fbVoter1Button(stColor := fbVoter1.fbStatusColor, nActiveTab := eActiveTab, sActiveName := sActiveName);
fbVoter2Button(stColor := fbVoter2.fbStatusColor, nActiveTab := eActiveTab, sActiveName := sActiveName);
fbVoter3Button(stColor := fbVoter3.fbStatusColor, nActiveTab := eActiveTab, sActiveName := sActiveName);
fbVoter4Button(stColor := fbVoter4.fbStatusColor, nActiveTab := eActiveTab, sActiveName := sActiveName);
fbVoter5Button(stColor := fbVoter5.fbStatusColor, nActiveTab := eActiveTab, sActiveName := sActiveName);
fbVoter6Button(stColor := fbVoter6.fbStatusColor, nActiveTab := eActiveTab, sActiveName := sActiveName);
fbVoter7Button(stColor := fbVoter7.fbStatusColor, nActiveTab := eActiveTab, sActiveName := sActiveName);
fbVoter8Button(stColor := fbVoter8.fbStatusColor, nActiveTab := eActiveTab, sActiveName := sActiveName);
fbVoter9Button(stColor := fbVoter9.fbStatusColor, nActiveTab := eActiveTab, sActiveName := sActiveName);
fbVoter10Button(stColor := fbVoter10.fbStatusColor, nActiveTab := eActiveTab, sActiveName := sActiveName);
    
M_UpdateStatusColor();

END_FUNCTION_BLOCK

// HMI/POUs/Subsystems/IMG/FB_HMI_IMG
FUNCTION_BLOCK FB_HMI_IMG EXTENDS FB_HMI_COMPONENT
VAR_INPUT
    bConnected : BOOL;
END_VAR
VAR_OUTPUT
END_VAR
VAR_IN_OUT
    temperatures    : FB_METIS_TEMPERATURES;
    heaters         : FB_METIS_HEATERS;
    voters          : FB_METIS_VOTERS;
    tctrl           : FB_METIS_TCTRL;
    lakeshores      : FB_METIS_LAKESHORES;
END_VAR
VAR
    // active tab of the main frame
    eActiveTab : E_HMI_IMG_TABS := E_HMI_IMG_TABS.TEMPERATURES;
    sActiveName : STRING;
    
    // components
    fbTemperatures : FB_HMI_IMG_TEMPERATURES;
    fbVoters       : FB_HMI_IMG_VOTERS;
    fbTControl     : FB_HMI_IMG_TCTRL;
    fbHeaters      : FB_HMI_IMG_HEATERS;
    fbLakeshoreLm  : FB_HMI_LAKESHORE;
    fbLakeshoreN   : FB_HMI_LAKESHORE;
    
    // buttons
    fbTemperaturesButton : FB_HMI_BUTTON(sName := 'Temperatures'         , sIconName := '', nThisTab := E_HMI_IMG_TABS.TEMPERATURES);
    fbVotersButton       : FB_HMI_BUTTON(sName := 'Voters'               , sIconName := '', nThisTab := E_HMI_IMG_TABS.VOTERS);
    fbHeatersButton      : FB_HMI_BUTTON(sName := 'Heaters'              , sIconName := '', nThisTab := E_HMI_IMG_TABS.HEATERS);
    fbLakeshoreLmButton  : FB_HMI_BUTTON(sName := 'Lakeshore LM'         , sIconName := '', nThisTab := E_HMI_IMG_TABS.LAKESHORE_LM_DET);
    fbLakeshoreNButton   : FB_HMI_BUTTON(sName := 'Lakeshore N'          , sIconName := '', nThisTab := E_HMI_IMG_TABS.LAKESHORE_N_DET);
    fbTControlButton     : FB_HMI_BUTTON(sName := 'Control loops'        , sIconName := '', nThisTab := E_HMI_IMG_TABS.TCONTROL);
    
    // connection status
    sConnected           : STRING;
    eConnectedColor      : E_HMI_COLORS;
END_VAR

// update the connection status
sConnected      := F_GetConnectionString(bConnected);
eConnectedColor := F_GetConnectionColor(bConnected); 

// update the components
fbTemperatures(fbInstance := temperatures, bConnected := bConnected);
fbVoters(fbInstance := voters, bConnected := bConnected);
fbTControl(fbInstance := tctrl, bConnected := bConnected);
fbHeaters(fbInstance := heaters, bConnected := bConnected);
fbLakeshoreLm(fbInstance := lakeshores.ls_img_lm, bConnected := bConnected);
fbLakeshoreN(fbInstance := lakeshores.ls_img_n, bConnected := bConnected);


// update the buttons
// sca
fbTemperaturesButton(
    stColor     := fbTemperatures.fbStatusColor,
    nActiveTab  := eActiveTab,
    sActiveName := sActiveName);
fbVotersButton(
    stColor     := fbVoters.fbStatusColor,
    nActiveTab  := eActiveTab,
    sActiveName := sActiveName);
fbHeatersButton(
    stColor     := fbHeaters.fbStatusColor,
    nActiveTab  := eActiveTab,
    sActiveName := sActiveName);
fbLakeshoreLmButton(
    stColor     := fbLakeshoreLm.fbStatusColor,
    nActiveTab  := eActiveTab,
    sActiveName := sActiveName);
fbLakeshoreNButton(
    stColor     := fbLakeshoreN.fbStatusColor,
    nActiveTab  := eActiveTab,
    sActiveName := sActiveName);
fbTControlButton(
    stColor     := fbTControl.fbStatusColor,
    nActiveTab  := eActiveTab,
    sActiveName := sActiveName);

// update the summary health/busy status
fbHealthStatus(
    bIsEnabled  := bConnected,
    bIsGood     :=     fbTemperatures.fbHealthStatus.bGood
                   AND fbVoters.fbHealthStatus.bGood
                   AND fbTControl.fbHealthStatus.bGood
                   AND fbHeaters.fbHealthStatus.bGood
                   AND fbLakeshoreLm.fbHealthStatus.bGood
                   AND fbLakeshoreN.fbHealthStatus.bGood,
    bHasWarning :=     fbTemperatures.fbHealthStatus.bWarning
                    OR fbVoters.fbHealthStatus.bWarning
                    OR fbTControl.fbHealthStatus.bWarning
                    OR fbHeaters.fbHealthStatus.bWarning
                    OR fbLakeshoreLm.fbHealthStatus.bWarning
                    OR fbLakeshoreN.fbHealthStatus.bWarning);

fbBusyStatus(
    bIsEnabled   := bConnected,
    bIsBusy      :=    fbTemperatures.fbBusyStatus.bBusy
                    OR fbVoters.fbBusyStatus.bBusy
                    OR fbTControl.fbBusyStatus.bBusy
                    OR fbHeaters.fbBusyStatus.bBusy
                    OR fbLakeshoreLm.fbBusyStatus.bBusy
                    OR fbLakeshoreN.fbBusyStatus.bBusy);

M_UpdateStatusColor();

END_FUNCTION_BLOCK

// HMI/POUs/Util/Functions/F_GetConnectionString
FUNCTION F_GetConnectionString : STRING
VAR_INPUT
    bConnected : BOOL;
END_VAR
VAR
END_VAR

IF bConnected THEN
    F_GetConnectionString := 'Connected';
ELSE
    F_GetConnectionString := 'Disconnected';
END_IF

END_FUNCTION

// HMI/POUs/Util/Functions/F_GetConnectionColor
FUNCTION F_GetConnectionColor : E_HMI_COLORS
VAR_INPUT
    bConnected : BOOL;
END_VAR
VAR
END_VAR

IF bConnected THEN
    F_GetConnectionColor := E_HMI_COLORS.GREEN;
ELSE
    F_GetConnectionColor := E_HMI_COLORS.RED;
END_IF

END_FUNCTION

// HMI/POUs/Subsystems/LMS/Components/FB_HMI_LMS_HEATERS
FUNCTION_BLOCK FB_HMI_LMS_HEATERS EXTENDS FB_HMI_COMPONENT
VAR_INPUT
END_VAR
VAR_OUTPUT
END_VAR
VAR_IN_OUT
    fbInstance : FB_METIS_HEATERS;
END_VAR
VAR
//    eActiveTab : E_HMI_CRY_HEATER_TABS;
//    sActiveName : STRING;
    
//    h_img_wuh_1_button  : FB_HMI_BUTTON(sName := 'H_IMG_WUH_1' , sIconName := '', nThisTab := E_HMI_IMG_HEATER_TABS.H_IMG_WUH_1);
//    h_img_wuh_2_button  : FB_HMI_BUTTON(sName := 'H_IMG_WUH_2' , sIconName := '', nThisTab := E_HMI_IMG_HEATER_TABS.H_IMG_WUH_2);
//    h_img_lmd_2_button  : FB_HMI_BUTTON(sName := 'H_IMG_LMD_2' , sIconName := '', nThisTab := E_HMI_IMG_HEATER_TABS.H_IMG_LMD_2);
//    h_img_lmp_2_button  : FB_HMI_BUTTON(sName := 'H_IMG_LMP_2' , sIconName := '', nThisTab := E_HMI_IMG_HEATER_TABS.H_IMG_LMP_2);
//    h_img_nd_2_button   : FB_HMI_BUTTON(sName := 'H_IMG_ND_2'  , sIconName := '', nThisTab := E_HMI_IMG_HEATER_TABS.H_IMG_ND_2);
    
//    h_img_wuh_1 : FB_HMI_METIS_HEATER;
//    h_img_wuh_2 : FB_HMI_METIS_HEATER;
//    h_img_lmd_2 : FB_HMI_METIS_HEATER;
//    h_img_lmp_2 : FB_HMI_METIS_HEATER;
//    h_img_nd_2  : FB_HMI_METIS_HEATER;
END_VAR

fbHealthStatus(bIsEnabled := FALSE);
fbBusyStatus(bIsEnabled := FALSE);

//fbHealthStatus(
//    bIsEnabled := TRUE,
//    bIsGood := NOT(    fbInstance.h_img_wuh_1.stat.bError
//                    OR fbInstance.h_img_wuh_2.stat.bError
//                    OR fbInstance.h_img_lmd_2.stat.bError
//                    OR fbInstance.h_img_lmp_2.stat.bError
//                    OR fbInstance.h_img_nd_2.stat.bError ),
//    bHasWarning := (    fbInstance.h_img_wuh_1.stat.bWarning
//                     OR fbInstance.h_img_wuh_2.stat.bWarning
//                     OR fbInstance.h_img_lmd_2.stat.bWarning
//                     OR fbInstance.h_img_lmp_2.stat.bWarning
//                     OR fbInstance.h_img_nd_2.stat.bWarning));

//fbBusyStatus(
//    bIsEnabled := TRUE,
//    bIsBusy := FALSE);

//h_img_wuh_1(fbInstance := fbInstance.h_img_wuh_1);
//h_img_wuh_2(fbInstance := fbInstance.h_img_wuh_2);
//h_img_lmd_2(fbInstance := fbInstance.h_img_lmd_2);
//h_img_lmp_2(fbInstance := fbInstance.h_img_lmp_2);
//h_img_nd_2(fbInstance := fbInstance.h_img_nd_2);

//h_img_wuh_1_button(stColor := h_img_wuh_1.fbStatusColor, nActiveTab := eActiveTab, sActiveName := sActiveName);
//h_img_wuh_2_button(stColor := h_img_wuh_2.fbStatusColor, nActiveTab := eActiveTab, sActiveName := sActiveName);
//h_img_lmd_2_button(stColor := h_img_lmd_2.fbStatusColor, nActiveTab := eActiveTab, sActiveName := sActiveName);
//h_img_lmp_2_button(stColor := h_img_lmp_2.fbStatusColor, nActiveTab := eActiveTab, sActiveName := sActiveName);
//h_img_nd_2_button(stColor := h_img_nd_2.fbStatusColor, nActiveTab := eActiveTab, sActiveName := sActiveName);

M_UpdateStatusColor();

END_FUNCTION_BLOCK

// HMI/POUs/Subsystems/LMS/Components/FB_HMI_LMS_TCTRL
FUNCTION_BLOCK FB_HMI_LMS_TCTRL EXTENDS FB_HMI_COMPONENT
VAR_INPUT
END_VAR
VAR_OUTPUT
END_VAR
VAR_IN_OUT
    fbInstance : FB_METIS_TCTRL;
END_VAR
VAR
//    eActiveTab : E_HMI_IMG_TC_TABS;
//    sActiveName : STRING;
    
//    tc_img_wuh_1_button  : FB_HMI_BUTTON(sName := 'TC_IMG_WUH_1' , sIconName := '', nThisTab := E_HMI_IMG_TC_TABS.TC_IMG_WUH_1);
//    tc_img_wuh_2_button  : FB_HMI_BUTTON(sName := 'TC_IMG_WUH_2' , sIconName := '', nThisTab := E_HMI_IMG_TC_TABS.TC_IMG_WUH_2);
//    tc_img_lmd_2_button  : FB_HMI_BUTTON(sName := 'TC_IMG_LMD_2' , sIconName := '', nThisTab := E_HMI_IMG_TC_TABS.TC_IMG_LMD_2);
//    tc_img_lmp_2_button  : FB_HMI_BUTTON(sName := 'TC_IMG_LMP_2' , sIconName := '', nThisTab := E_HMI_IMG_TC_TABS.TC_IMG_LMP_2);
//    tc_img_nd_2_button   : FB_HMI_BUTTON(sName := 'TC_IMG_ND_2'  , sIconName := '', nThisTab := E_HMI_IMG_TC_TABS.TC_IMG_ND_2);
    
//    tc_img_wuh_1 : FB_HMI_METIS_CTRL_DT670;
//    tc_img_wuh_2 : FB_HMI_METIS_CTRL_DT670;
//    tc_img_lmd_2 : FB_HMI_METIS_CTRL_DT670;
//    tc_img_lmp_2 : FB_HMI_METIS_CTRL_DT670;
//    tc_img_nd_2  : FB_HMI_METIS_CTRL_DT670;
END_VAR

fbHealthStatus(bIsEnabled := FALSE);
fbBusyStatus(bIsEnabled := FALSE);

//fbHealthStatus(
//    bIsEnabled := TRUE,
//    bIsGood := NOT(    fbInstance.tc_img_wuh_1.stat.bError
//                    OR fbInstance.tc_img_wuh_2.stat.bError
//                    OR fbInstance.tc_img_lmd_2.stat.bError
//                    OR fbInstance.tc_img_lmp_2.stat.bError
//                    OR fbInstance.tc_img_nd_2.stat.bError ),
//    bHasWarning := (    fbInstance.tc_img_wuh_1.stat.bWarning
//                     OR fbInstance.tc_img_wuh_2.stat.bWarning
//                     OR fbInstance.tc_img_lmd_2.stat.bWarning
//                     OR fbInstance.tc_img_lmp_2.stat.bWarning
//                     OR fbInstance.tc_img_nd_2.stat.bWarning));

//tc_img_wuh_1(fbInstance := fbInstance.tc_img_wuh_1);
//tc_img_wuh_2(fbInstance := fbInstance.tc_img_wuh_2);
//tc_img_lmd_2(fbInstance := fbInstance.tc_img_lmd_2);
//tc_img_lmp_2(fbInstance := fbInstance.tc_img_lmp_2);
//tc_img_nd_2(fbInstance := fbInstance.tc_img_nd_2);

//tc_img_wuh_1_button(stColor := tc_img_wuh_1.fbStatusColor, nActiveTab := eActiveTab, sActiveName := sActiveName);
//tc_img_wuh_2_button(stColor := tc_img_wuh_2.fbStatusColor, nActiveTab := eActiveTab, sActiveName := sActiveName);
//tc_img_lmd_2_button(stColor := tc_img_lmd_2.fbStatusColor, nActiveTab := eActiveTab, sActiveName := sActiveName);
//tc_img_lmp_2_button(stColor := tc_img_lmp_2.fbStatusColor, nActiveTab := eActiveTab, sActiveName := sActiveName);
//tc_img_nd_2_button(stColor := tc_img_nd_2.fbStatusColor, nActiveTab := eActiveTab, sActiveName := sActiveName);

//fbBusyStatus(
//    bIsEnabled := TRUE,
//    bIsBusy := FALSE);

M_UpdateStatusColor();

END_FUNCTION_BLOCK

// HMI/POUs/Subsystems/LMS/Components/FB_HMI_LMS_TEMPERATURES
FUNCTION_BLOCK FB_HMI_LMS_TEMPERATURES EXTENDS FB_HMI_COMPONENT
VAR_INPUT
END_VAR
VAR_OUTPUT
END_VAR
VAR_IN_OUT
    fbInstance : FB_METIS_TEMPERATURES;
END_VAR
VAR
END_VAR

fbHealthStatus(bIsEnabled := FALSE);
fbBusyStatus(bIsEnabled := FALSE);

//fbHealthStatus(
//    bIsEnabled := TRUE,
//    bIsGood :=     fbInstance.t_img_lpw_1.stat.bValid
//               AND fbInstance.t_img_lpw_2.stat.bValid
//               AND fbInstance.t_img_lfw_1.stat.bValid
//               AND fbInstance.t_img_lfw_2.stat.bValid
//               AND fbInstance.t_img_lpr_1.stat.bValid
//               AND fbInstance.t_img_bwu_3.stat.bValid
//               AND fbInstance.t_img_lnd_1.stat.bValid
//               AND fbInstance.t_img_lnd_2.stat.bValid
//               AND fbInstance.t_img_npw_1.stat.bValid
//               AND fbInstance.t_img_npw_2.stat.bValid
//               AND fbInstance.t_img_nfw_1.stat.bValid
//               AND fbInstance.t_img_nfw_2.stat.bValid
//               AND fbInstance.t_img_npr_1.stat.bValid
//               AND fbInstance.t_img_bwu_2.stat.bValid
//               AND fbInstance.t_img_nnd_1.stat.bValid
//               AND fbInstance.t_img_nnd_2.stat.bValid
//               AND fbInstance.t_img_opt_1.stat.bValid
//               AND fbInstance.t_img_bwu_1.stat.bValid
//               AND fbInstance.t_img_ctr_1.stat.bValid
//               AND fbInstance.t_img_ctr_2.stat.bValid
//               AND fbInstance.t_img_70k_1.stat.bValid
//               AND fbInstance.t_img_ln2_1.stat.bValid
//               AND fbInstance.t_img_ln2_2.stat.bValid
//               AND fbInstance.t_img_hex_1.stat.bValid
//               AND fbInstance.t_img_lmd_1.stat.bValid
//               AND fbInstance.t_img_lmd_2.stat.bValid
//               AND fbInstance.t_img_lmp_1.stat.bValid
//               AND fbInstance.t_img_lmp_2.stat.bValid
//               AND fbInstance.t_img_nd_1.stat.bValid
//               AND fbInstance.t_img_nd_2.stat.bValid,
//    bHasWarning := (    fbInstance.t_img_lpw_1.stat.bWarning
//                     OR fbInstance.t_img_lpw_2.stat.bWarning
//                     OR fbInstance.t_img_lfw_1.stat.bWarning
//                     OR fbInstance.t_img_lfw_2.stat.bWarning
//                     OR fbInstance.t_img_lpr_1.stat.bWarning
//                     OR fbInstance.t_img_bwu_3.stat.bWarning
//                     OR fbInstance.t_img_lnd_1.stat.bWarning
//                     OR fbInstance.t_img_lnd_2.stat.bWarning
//                     OR fbInstance.t_img_npw_1.stat.bWarning
//                     OR fbInstance.t_img_npw_2.stat.bWarning
//                     OR fbInstance.t_img_nfw_1.stat.bWarning
//                     OR fbInstance.t_img_nfw_2.stat.bWarning
//                     OR fbInstance.t_img_npr_1.stat.bWarning
//                     OR fbInstance.t_img_bwu_2.stat.bWarning
//                     OR fbInstance.t_img_nnd_1.stat.bWarning
//                     OR fbInstance.t_img_nnd_2.stat.bWarning
//                     OR fbInstance.t_img_opt_1.stat.bWarning
//                     OR fbInstance.t_img_bwu_1.stat.bWarning
//                     OR fbInstance.t_img_ctr_1.stat.bWarning
//                     OR fbInstance.t_img_ctr_2.stat.bWarning
//                     OR fbInstance.t_img_ln2_1.stat.bWarning
//                     OR fbInstance.t_img_ln2_1.stat.bWarning
//                     OR fbInstance.t_img_ln2_2.stat.bWarning
//                     OR fbInstance.t_img_hex_1.stat.bWarning
//                     OR fbInstance.t_img_lmd_1.stat.bWarning
//                     OR fbInstance.t_img_lmd_2.stat.bWarning
//                     OR fbInstance.t_img_lmp_1.stat.bWarning
//                     OR fbInstance.t_img_lmp_2.stat.bWarning
//                     OR fbInstance.t_img_nd_1.stat.bWarning
//                     OR fbInstance.t_img_nd_2.stat.bWarning));
                     
//fbBusyStatus(
//    bIsEnabled := TRUE,
//    bIsBusy := FALSE);

M_UpdateStatusColor();

END_FUNCTION_BLOCK

// HMI/POUs/Subsystems/LMS/Components/FB_HMI_LMS_VOTERS
FUNCTION_BLOCK FB_HMI_LMS_VOTERS EXTENDS FB_HMI_COMPONENT
VAR_INPUT
END_VAR
VAR_OUTPUT
END_VAR
VAR_IN_OUT
    fbInstance : FB_METIS_VOTERS;
END_VAR
VAR
    eActiveTab : E_HMI_VOTER_TABS;
    sActiveName : STRING;
    
    fbVoter1Button  : FB_HMI_BUTTON(sName := 'Voter 1' , sIconName := '', nThisTab := E_HMI_VOTER_TABS.VOTER_1);
    fbVoter2Button  : FB_HMI_BUTTON(sName := 'Voter 2' , sIconName := '', nThisTab := E_HMI_VOTER_TABS.VOTER_2);
    fbVoter3Button  : FB_HMI_BUTTON(sName := 'Voter 3' , sIconName := '', nThisTab := E_HMI_VOTER_TABS.VOTER_3);
    fbVoter4Button  : FB_HMI_BUTTON(sName := 'Voter 4' , sIconName := '', nThisTab := E_HMI_VOTER_TABS.VOTER_4);
    fbVoter5Button  : FB_HMI_BUTTON(sName := 'Voter 5' , sIconName := '', nThisTab := E_HMI_VOTER_TABS.VOTER_5);
    fbVoter6Button  : FB_HMI_BUTTON(sName := 'Voter 6' , sIconName := '', nThisTab := E_HMI_VOTER_TABS.VOTER_6);
    fbVoter7Button  : FB_HMI_BUTTON(sName := 'Voter 7' , sIconName := '', nThisTab := E_HMI_VOTER_TABS.VOTER_7);
    fbVoter8Button  : FB_HMI_BUTTON(sName := 'Voter 8' , sIconName := '', nThisTab := E_HMI_VOTER_TABS.VOTER_8);
    fbVoter9Button  : FB_HMI_BUTTON(sName := 'Voter 9' , sIconName := '', nThisTab := E_HMI_VOTER_TABS.VOTER_9);
    fbVoter10Button : FB_HMI_BUTTON(sName := 'Voter 10', sIconName := '', nThisTab := E_HMI_VOTER_TABS.VOTER_10);
    
    fbVoter1 : FB_HMI_VOTER;
    fbVoter2 : FB_HMI_VOTER;
    fbVoter3 : FB_HMI_VOTER;
    fbVoter4 : FB_HMI_VOTER;
    fbVoter5 : FB_HMI_VOTER;
    fbVoter6 : FB_HMI_VOTER;
    fbVoter7 : FB_HMI_VOTER;
    fbVoter8 : FB_HMI_VOTER;
    fbVoter9 : FB_HMI_VOTER;
    fbVoter10 : FB_HMI_VOTER;
END_VAR

fbHealthStatus(bIsEnabled := FALSE);
fbBusyStatus(bIsEnabled := FALSE);

//fbHealthStatus(
//    bIsEnabled :=  fbVoter1.fbHealthStatus.bEnabled
//                OR fbVoter2.fbHealthStatus.bEnabled
//                OR fbVoter3.fbHealthStatus.bEnabled
//                OR fbVoter4.fbHealthStatus.bEnabled
//                OR fbVoter5.fbHealthStatus.bEnabled
//                OR fbVoter6.fbHealthStatus.bEnabled
//                OR fbVoter7.fbHealthStatus.bEnabled
//                OR fbVoter8.fbHealthStatus.bEnabled
//                OR fbVoter9.fbHealthStatus.bEnabled
//                OR fbVoter10.fbHealthStatus.bEnabled,
//    bIsGood :=  (fbVoter1.fbHealthStatus.bGood OR NOT fbVoter1.fbHealthStatus.bEnabled)
//            AND (fbVoter2.fbHealthStatus.bGood OR NOT fbVoter2.fbHealthStatus.bEnabled)
//            AND (fbVoter3.fbHealthStatus.bGood OR NOT fbVoter3.fbHealthStatus.bEnabled)
//            AND (fbVoter4.fbHealthStatus.bGood OR NOT fbVoter4.fbHealthStatus.bEnabled)
//            AND (fbVoter5.fbHealthStatus.bGood OR NOT fbVoter5.fbHealthStatus.bEnabled)
//            AND (fbVoter6.fbHealthStatus.bGood OR NOT fbVoter6.fbHealthStatus.bEnabled)
//            AND (fbVoter7.fbHealthStatus.bGood OR NOT fbVoter7.fbHealthStatus.bEnabled)
//            AND (fbVoter8.fbHealthStatus.bGood OR NOT fbVoter8.fbHealthStatus.bEnabled)
//            AND (fbVoter9.fbHealthStatus.bGood OR NOT fbVoter9.fbHealthStatus.bEnabled)
//            AND (fbVoter10.fbHealthStatus.bGood OR NOT fbVoter10.fbHealthStatus.bEnabled));

//fbBusyStatus(
//    bIsEnabled := TRUE,
//    bIsBusy := FALSE);

//fbVoter1(fbInstance := fbInstance.vote_img_1);
//fbVoter2(fbInstance := fbInstance.vote_img_2);
//fbVoter3(fbInstance := fbInstance.vote_img_3);
//fbVoter4(fbInstance := fbInstance.vote_img_4);
//fbVoter5(fbInstance := fbInstance.vote_img_5);
//fbVoter6(fbInstance := fbInstance.vote_img_6);
//fbVoter7(fbInstance := fbInstance.vote_img_7);
//fbVoter8(fbInstance := fbInstance.vote_img_8);
//fbVoter9(fbInstance := fbInstance.vote_img_9);
//fbVoter10(fbInstance := fbInstance.vote_img_10);

//fbVoter1Button(stColor := fbVoter1.fbStatusColor, nActiveTab := eActiveTab, sActiveName := sActiveName);
//fbVoter2Button(stColor := fbVoter2.fbStatusColor, nActiveTab := eActiveTab, sActiveName := sActiveName);
//fbVoter3Button(stColor := fbVoter3.fbStatusColor, nActiveTab := eActiveTab, sActiveName := sActiveName);
//fbVoter4Button(stColor := fbVoter4.fbStatusColor, nActiveTab := eActiveTab, sActiveName := sActiveName);
//fbVoter5Button(stColor := fbVoter5.fbStatusColor, nActiveTab := eActiveTab, sActiveName := sActiveName);
//fbVoter6Button(stColor := fbVoter6.fbStatusColor, nActiveTab := eActiveTab, sActiveName := sActiveName);
//fbVoter7Button(stColor := fbVoter7.fbStatusColor, nActiveTab := eActiveTab, sActiveName := sActiveName);
//fbVoter8Button(stColor := fbVoter8.fbStatusColor, nActiveTab := eActiveTab, sActiveName := sActiveName);
//fbVoter9Button(stColor := fbVoter9.fbStatusColor, nActiveTab := eActiveTab, sActiveName := sActiveName);
//fbVoter10Button(stColor := fbVoter10.fbStatusColor, nActiveTab := eActiveTab, sActiveName := sActiveName);
    
M_UpdateStatusColor();

END_FUNCTION_BLOCK

// HMI/POUs/Subsystems/LMS/FB_HMI_LMS
FUNCTION_BLOCK FB_HMI_LMS EXTENDS FB_HMI_COMPONENT
VAR_INPUT
END_VAR
VAR_OUTPUT
END_VAR
VAR_IN_OUT
    temperatures    : FB_METIS_TEMPERATURES;
    heaters         : FB_METIS_HEATERS;
    voters          : FB_METIS_VOTERS;
    tctrl           : FB_METIS_TCTRL;
END_VAR
VAR
    // active tab of the main frame
    eActiveTab : E_HMI_LMS_TABS := E_HMI_LMS_TABS.TEMPERATURES;
    sActiveName : STRING;
    
    // components
    fbTemperatures : FB_HMI_LMS_TEMPERATURES;
    fbVoters       : FB_HMI_LMS_VOTERS;
    fbTControl     : FB_HMI_LMS_TCTRL;
    fbHeaters      : FB_HMI_LMS_HEATERS;
    
    // buttons
    fbTemperaturesButton : FB_HMI_BUTTON(sName := 'Temperatures'         , sIconName := '', nThisTab := E_HMI_LMS_TABS.TEMPERATURES);
    fbVotersButton       : FB_HMI_BUTTON(sName := 'Voters'               , sIconName := '', nThisTab := E_HMI_LMS_TABS.VOTERS);
    fbHeatersButton      : FB_HMI_BUTTON(sName := 'Heaters'              , sIconName := '', nThisTab := E_HMI_LMS_TABS.HEATERS);
    fbTControlButton     : FB_HMI_BUTTON(sName := 'Control loops'        , sIconName := '', nThisTab := E_HMI_LMS_TABS.TCONTROL);
END_VAR

// update the components
fbTemperatures(fbInstance := temperatures);
fbVoters(fbInstance := voters);
fbTControl(fbInstance := tctrl);
fbHeaters(fbInstance := heaters);

// update the buttons
fbTemperaturesButton(
    stColor     := fbTemperatures.fbStatusColor,
    nActiveTab  := eActiveTab,
    sActiveName := sActiveName);
fbVotersButton(
    stColor     := fbVoters.fbStatusColor,
    nActiveTab  := eActiveTab,
    sActiveName := sActiveName);
fbHeatersButton(
    stColor     := fbHeaters.fbStatusColor,
    nActiveTab  := eActiveTab,
    sActiveName := sActiveName);
fbTControlButton(
    stColor     := fbTControl.fbStatusColor,
    nActiveTab  := eActiveTab,
    sActiveName := sActiveName);


// update the summary health/busy status
fbHealthStatus(
    bIsEnabled  := TRUE,
    bIsGood     :=     fbTemperatures.fbHealthStatus.bGood
                   AND fbVoters.fbHealthStatus.bGood
                   AND fbTControl.fbHealthStatus.bGood
                   AND fbHeaters.fbHealthStatus.bGood,
    bHasWarning :=     fbTemperatures.fbHealthStatus.bWarning
                    OR fbVoters.fbHealthStatus.bWarning
                    OR fbTControl.fbHealthStatus.bWarning
                    OR fbHeaters.fbHealthStatus.bWarning);

fbBusyStatus(
    bIsEnabled   := TRUE,
    bIsBusy      :=    fbTemperatures.fbBusyStatus.bBusy
                    OR fbVoters.fbBusyStatus.bBusy
                    OR fbTControl.fbBusyStatus.bBusy
                    OR fbHeaters.fbBusyStatus.bBusy);

M_UpdateStatusColor();

END_FUNCTION_BLOCK

// HMI/POUs/Subsystems/SCA/Components/FB_HMI_SCA_HEATERS
FUNCTION_BLOCK FB_HMI_SCA_HEATERS EXTENDS FB_HMI_COMPONENT
VAR_INPUT
    bConnected : BOOL;
END_VAR
VAR_OUTPUT
END_VAR
VAR_IN_OUT
    fbInstance : FB_METIS_HEATERS;
END_VAR
VAR
    eActiveTab : E_HMI_SCA_HEATER_TABS;
    sActiveName : STRING;
    
    h_sca_wuh_1_button  : FB_HMI_BUTTON(sName := 'H_SCA_WUH_1' , sIconName := '', nThisTab := E_HMI_SCA_HEATER_TABS.H_SCA_WUH_1);
    h_sca_wuh_2_button  : FB_HMI_BUTTON(sName := 'H_SCA_WUH_2' , sIconName := '', nThisTab := E_HMI_SCA_HEATER_TABS.H_SCA_WUH_2);
    h_sca_det_2_button  : FB_HMI_BUTTON(sName := 'H_SCA_DET_2' , sIconName := '', nThisTab := E_HMI_SCA_HEATER_TABS.H_SCA_DET_2);
    h_sca_dhs_2_button  : FB_HMI_BUTTON(sName := 'H_SCA_DHS_2' , sIconName := '', nThisTab := E_HMI_SCA_HEATER_TABS.H_SCA_DHS_2);
    
    h_sca_wuh_1 : FB_HMI_METIS_HEATER;
    h_sca_wuh_2 : FB_HMI_METIS_HEATER;
    h_sca_det_2 : FB_HMI_METIS_HEATER;
    h_sca_dhs_2 : FB_HMI_METIS_HEATER;
END_VAR

fbHealthStatus(
    bIsEnabled := bConnected,
    bIsGood := NOT(    fbInstance.h_sca_wuh_1.stat.bError
                    OR fbInstance.h_sca_wuh_2.stat.bError
                    OR fbInstance.h_sca_det_2.stat.bError
                    OR fbInstance.h_sca_dhs_2.stat.bError ),
    bHasWarning := (    fbInstance.h_sca_wuh_1.stat.bWarning
                     OR fbInstance.h_sca_wuh_2.stat.bWarning
                     OR fbInstance.h_sca_det_2.stat.bWarning
                     OR fbInstance.h_sca_dhs_2.stat.bWarning));
                     
fbBusyStatus(
    bIsEnabled := bConnected,
    bIsBusy := FALSE);

h_sca_wuh_1(fbInstance := fbInstance.h_sca_wuh_1);
h_sca_wuh_2(fbInstance := fbInstance.h_sca_wuh_2);
h_sca_det_2(fbInstance := fbInstance.h_sca_det_2);
h_sca_dhs_2(fbInstance := fbInstance.h_sca_dhs_2);

h_sca_wuh_1_button(stColor := h_sca_wuh_1.fbStatusColor, nActiveTab := eActiveTab, sActiveName := sActiveName);
h_sca_wuh_2_button(stColor := h_sca_wuh_2.fbStatusColor, nActiveTab := eActiveTab, sActiveName := sActiveName);
h_sca_det_2_button(stColor := h_sca_det_2.fbStatusColor, nActiveTab := eActiveTab, sActiveName := sActiveName);
h_sca_dhs_2_button(stColor := h_sca_dhs_2.fbStatusColor, nActiveTab := eActiveTab, sActiveName := sActiveName);

M_UpdateStatusColor();

END_FUNCTION_BLOCK

// HMI/POUs/Subsystems/SCA/Components/FB_HMI_SCA_TCTRL
FUNCTION_BLOCK FB_HMI_SCA_TCTRL EXTENDS FB_HMI_COMPONENT
VAR_INPUT
    bConnected : BOOL;
END_VAR
VAR_OUTPUT
END_VAR
VAR_IN_OUT
    fbInstance : FB_METIS_TCTRL;
END_VAR
VAR
    eActiveTab : E_HMI_SCA_TC_TABS;
    sActiveName : STRING;
    
    tc_sca_wuh_button    : FB_HMI_BUTTON(sName := 'TC_SCA_WUH'   , sIconName := '', nThisTab := E_HMI_SCA_TC_TABS.TC_SCA_WUH);
    tc_sca_det_2_button  : FB_HMI_BUTTON(sName := 'TC_SCA_DET_2' , sIconName := '', nThisTab := E_HMI_SCA_TC_TABS.TC_SCA_DET_2);
    tc_sca_dhs_2_button  : FB_HMI_BUTTON(sName := 'TC_SCA_DHS_2' , sIconName := '', nThisTab := E_HMI_SCA_TC_TABS.TC_SCA_DHS_2);
    
    tc_sca_wuh   : FB_HMI_METIS_CTRL_TEMPERATURE;
    tc_sca_det_2 : FB_HMI_METIS_CTRL_TEMPERATURE;
    tc_sca_dhs_2 : FB_HMI_METIS_CTRL_TEMPERATURE;
END_VAR

fbHealthStatus(
    bIsEnabled := bConnected,
    bIsGood := NOT(    fbInstance.tc_sca_wuh.stat.bError
                    OR fbInstance.tc_sca_det_2.stat.bError
                    OR fbInstance.tc_sca_dhs_2.stat.bError),
    bHasWarning := (    fbInstance.tc_sca_wuh.stat.bWarning
                     OR fbInstance.tc_sca_det_2.stat.bWarning
                     OR fbInstance.tc_sca_dhs_2.stat.bWarning));

tc_sca_wuh(  fbInstance := fbInstance.tc_sca_wuh);
tc_sca_det_2(fbInstance := fbInstance.tc_sca_det_2);
tc_sca_dhs_2(fbInstance := fbInstance.tc_sca_dhs_2);

tc_sca_wuh_button(stColor := tc_sca_wuh.fbStatusColor, nActiveTab := eActiveTab, sActiveName := sActiveName);
tc_sca_det_2_button(stColor := tc_sca_det_2.fbStatusColor, nActiveTab := eActiveTab, sActiveName := sActiveName);
tc_sca_dhs_2_button(stColor := tc_sca_dhs_2.fbStatusColor, nActiveTab := eActiveTab, sActiveName := sActiveName);


fbBusyStatus(
    bIsEnabled := bConnected,
    bIsBusy := FALSE);

M_UpdateStatusColor();

END_FUNCTION_BLOCK

// HMI/POUs/Subsystems/SCA/Components/FB_HMI_SCA_TEMPERATURES
FUNCTION_BLOCK FB_HMI_SCA_TEMPERATURES EXTENDS FB_HMI_COMPONENT
VAR_INPUT
    bConnected : BOOL;
END_VAR
VAR_OUTPUT
END_VAR
VAR_IN_OUT
    fbInstance : FB_METIS_TEMPERATURES;
END_VAR
VAR
END_VAR

fbHealthStatus(
    bIsEnabled := bConnected,
    bIsGood :=     fbInstance.t_sca_fw_1.stat.bValid
               AND fbInstance.t_sca_fw_2.stat.bValid
               AND fbInstance.t_sca_lu_1.stat.bValid
               AND fbInstance.t_sca_fm.stat.bValid
               AND fbInstance.t_sca_fs.stat.bValid
               AND fbInstance.t_sca_lu_2.stat.bValid
               AND fbInstance.t_sca_mod.stat.bValid
               AND fbInstance.t_sca_pyr.stat.bValid
               AND fbInstance.t_sca_h_1.stat.bValid
               AND fbInstance.t_sca_if_1.stat.bValid
               AND fbInstance.t_sca_if_2.stat.bValid
               AND fbInstance.t_sca_lu_1.stat.bValid
               AND fbInstance.t_sca_bp_1.stat.bValid
               AND fbInstance.t_sca_bp_2.stat.bValid
               AND fbInstance.t_sca_bp_3.stat.bValid
               AND fbInstance.t_sca_h_2.stat.bValid
               AND fbInstance.t_sca_det_1.stat.bValid
               AND fbInstance.t_sca_det_2.stat.bValid
               AND fbInstance.t_sca_dhs_1.stat.bValid
               AND fbInstance.t_sca_dhs_2.stat.bValid,
    bHasWarning := (    fbInstance.t_sca_fw_1.stat.bWarning
                     OR fbInstance.t_sca_fw_2.stat.bWarning
                     OR fbInstance.t_sca_lu_1.stat.bWarning
                     OR fbInstance.t_sca_fm.stat.bWarning
                     OR fbInstance.t_sca_fs.stat.bWarning
                     OR fbInstance.t_sca_lu_2.stat.bWarning
                     OR fbInstance.t_sca_mod.stat.bWarning
                     OR fbInstance.t_sca_pyr.stat.bWarning
                     OR fbInstance.t_sca_h_1.stat.bWarning
                     OR fbInstance.t_sca_if_1.stat.bWarning
                     OR fbInstance.t_sca_if_2.stat.bWarning
                     OR fbInstance.t_sca_lu_1.stat.bWarning
                     OR fbInstance.t_sca_bp_1.stat.bWarning
                     OR fbInstance.t_sca_bp_2.stat.bWarning
                     OR fbInstance.t_sca_bp_3.stat.bWarning
                     OR fbInstance.t_sca_h_2.stat.bWarning
                     OR fbInstance.t_sca_det_1.stat.bWarning
                     OR fbInstance.t_sca_det_2.stat.bWarning
                     OR fbInstance.t_sca_dhs_1.stat.bWarning
                     OR fbInstance.t_sca_dhs_2.stat.bWarning));
                     
fbBusyStatus(
    bIsEnabled := bConnected,
    bIsBusy := FALSE);

M_UpdateStatusColor();

END_FUNCTION_BLOCK

// HMI/POUs/Subsystems/SCA/Components/FB_HMI_SCA_VOTERS
FUNCTION_BLOCK FB_HMI_SCA_VOTERS EXTENDS FB_HMI_COMPONENT
VAR_INPUT
    bConnected : BOOL;
END_VAR
VAR_OUTPUT
END_VAR
VAR_IN_OUT
    fbInstance : FB_METIS_VOTERS;
END_VAR
VAR
    eActiveTab : E_HMI_VOTER_TABS;
    sActiveName : STRING;
    
    fbVoter1Button  : FB_HMI_BUTTON(sName := 'Voter 1' , sIconName := '', nThisTab := E_HMI_VOTER_TABS.VOTER_1);
    fbVoter2Button  : FB_HMI_BUTTON(sName := 'Voter 2' , sIconName := '', nThisTab := E_HMI_VOTER_TABS.VOTER_2);
    fbVoter3Button  : FB_HMI_BUTTON(sName := 'Voter 3' , sIconName := '', nThisTab := E_HMI_VOTER_TABS.VOTER_3);
    fbVoter4Button  : FB_HMI_BUTTON(sName := 'Voter 4' , sIconName := '', nThisTab := E_HMI_VOTER_TABS.VOTER_4);
    fbVoter5Button  : FB_HMI_BUTTON(sName := 'Voter 5' , sIconName := '', nThisTab := E_HMI_VOTER_TABS.VOTER_5);
    fbVoter6Button  : FB_HMI_BUTTON(sName := 'Voter 6' , sIconName := '', nThisTab := E_HMI_VOTER_TABS.VOTER_6);
    fbVoter7Button  : FB_HMI_BUTTON(sName := 'Voter 7' , sIconName := '', nThisTab := E_HMI_VOTER_TABS.VOTER_7);
    fbVoter8Button  : FB_HMI_BUTTON(sName := 'Voter 8' , sIconName := '', nThisTab := E_HMI_VOTER_TABS.VOTER_8);
    fbVoter9Button  : FB_HMI_BUTTON(sName := 'Voter 9' , sIconName := '', nThisTab := E_HMI_VOTER_TABS.VOTER_9);
    fbVoter10Button : FB_HMI_BUTTON(sName := 'Voter 10', sIconName := '', nThisTab := E_HMI_VOTER_TABS.VOTER_10);
    
    fbVoter1 : FB_HMI_VOTER;
    fbVoter2 : FB_HMI_VOTER;
    fbVoter3 : FB_HMI_VOTER;
    fbVoter4 : FB_HMI_VOTER;
    fbVoter5 : FB_HMI_VOTER;
    fbVoter6 : FB_HMI_VOTER;
    fbVoter7 : FB_HMI_VOTER;
    fbVoter8 : FB_HMI_VOTER;
    fbVoter9 : FB_HMI_VOTER;
    fbVoter10 : FB_HMI_VOTER;
END_VAR

fbHealthStatus(
    bIsEnabled := bConnected AND (
                   fbVoter1.fbHealthStatus.bEnabled
                OR fbVoter2.fbHealthStatus.bEnabled
                OR fbVoter3.fbHealthStatus.bEnabled
                OR fbVoter4.fbHealthStatus.bEnabled
                OR fbVoter5.fbHealthStatus.bEnabled
                OR fbVoter6.fbHealthStatus.bEnabled
                OR fbVoter7.fbHealthStatus.bEnabled
                OR fbVoter8.fbHealthStatus.bEnabled
                OR fbVoter9.fbHealthStatus.bEnabled
                OR fbVoter10.fbHealthStatus.bEnabled),
    bIsGood :=  (fbVoter1.fbHealthStatus.bGood OR NOT fbVoter1.fbHealthStatus.bEnabled)
            AND (fbVoter2.fbHealthStatus.bGood OR NOT fbVoter2.fbHealthStatus.bEnabled)
            AND (fbVoter3.fbHealthStatus.bGood OR NOT fbVoter3.fbHealthStatus.bEnabled)
            AND (fbVoter4.fbHealthStatus.bGood OR NOT fbVoter4.fbHealthStatus.bEnabled)
            AND (fbVoter5.fbHealthStatus.bGood OR NOT fbVoter5.fbHealthStatus.bEnabled)
            AND (fbVoter6.fbHealthStatus.bGood OR NOT fbVoter6.fbHealthStatus.bEnabled)
            AND (fbVoter7.fbHealthStatus.bGood OR NOT fbVoter7.fbHealthStatus.bEnabled)
            AND (fbVoter8.fbHealthStatus.bGood OR NOT fbVoter8.fbHealthStatus.bEnabled)
            AND (fbVoter9.fbHealthStatus.bGood OR NOT fbVoter9.fbHealthStatus.bEnabled)
            AND (fbVoter10.fbHealthStatus.bGood OR NOT fbVoter10.fbHealthStatus.bEnabled));

fbBusyStatus(
    bIsEnabled := bConnected,
    bIsBusy := FALSE);

fbVoter1(fbInstance := fbInstance.vote_sca_1);
fbVoter2(fbInstance := fbInstance.vote_sca_2);
fbVoter3(fbInstance := fbInstance.vote_sca_3);
fbVoter4(fbInstance := fbInstance.vote_sca_4);
fbVoter5(fbInstance := fbInstance.vote_sca_5);
fbVoter6(fbInstance := fbInstance.vote_sca_6);
fbVoter7(fbInstance := fbInstance.vote_sca_7);
fbVoter8(fbInstance := fbInstance.vote_sca_8);
fbVoter9(fbInstance := fbInstance.vote_sca_9);
fbVoter10(fbInstance := fbInstance.vote_sca_10);

fbVoter1Button(stColor := fbVoter1.fbStatusColor, nActiveTab := eActiveTab, sActiveName := sActiveName);
fbVoter2Button(stColor := fbVoter2.fbStatusColor, nActiveTab := eActiveTab, sActiveName := sActiveName);
fbVoter3Button(stColor := fbVoter3.fbStatusColor, nActiveTab := eActiveTab, sActiveName := sActiveName);
fbVoter4Button(stColor := fbVoter4.fbStatusColor, nActiveTab := eActiveTab, sActiveName := sActiveName);
fbVoter5Button(stColor := fbVoter5.fbStatusColor, nActiveTab := eActiveTab, sActiveName := sActiveName);
fbVoter6Button(stColor := fbVoter6.fbStatusColor, nActiveTab := eActiveTab, sActiveName := sActiveName);
fbVoter7Button(stColor := fbVoter7.fbStatusColor, nActiveTab := eActiveTab, sActiveName := sActiveName);
fbVoter8Button(stColor := fbVoter8.fbStatusColor, nActiveTab := eActiveTab, sActiveName := sActiveName);
fbVoter9Button(stColor := fbVoter9.fbStatusColor, nActiveTab := eActiveTab, sActiveName := sActiveName);
fbVoter10Button(stColor := fbVoter10.fbStatusColor, nActiveTab := eActiveTab, sActiveName := sActiveName);
    
M_UpdateStatusColor();

END_FUNCTION_BLOCK

// HMI/POUs/Subsystems/SCA/FB_HMI_SCA
FUNCTION_BLOCK FB_HMI_SCA EXTENDS FB_HMI_COMPONENT
VAR_INPUT
    bConnected : BOOL;
END_VAR
VAR_OUTPUT
END_VAR
VAR_IN_OUT
    temperatures    : FB_METIS_TEMPERATURES;
    heaters         : FB_METIS_HEATERS;
    voters          : FB_METIS_VOTERS;
    tctrl           : FB_METIS_TCTRL;
    lakeshores      : FB_METIS_LAKESHORES;
END_VAR
VAR
    // active tab of the main frame
    eActiveTab : E_HMI_SCA_TABS := E_HMI_SCA_TABS.TEMPERATURES;
    sActiveName : STRING;
    
    // components
    fbTemperatures : FB_HMI_SCA_TEMPERATURES;
    fbVoters       : FB_HMI_SCA_VOTERS;
    fbTControl     : FB_HMI_SCA_TCTRL;
    fbHeaters      : FB_HMI_SCA_HEATERS;
    fbLakeshore    : FB_HMI_LAKESHORE;
    
    fbTemperaturesButton : FB_HMI_BUTTON(sName := 'Temperatures'         , sIconName := '', nThisTab := E_HMI_SCA_TABS.TEMPERATURES);
    fbVotersButton       : FB_HMI_BUTTON(sName := 'Voters'               , sIconName := '', nThisTab := E_HMI_SCA_TABS.VOTERS);
    fbHeatersButton      : FB_HMI_BUTTON(sName := 'Heaters'              , sIconName := '', nThisTab := E_HMI_SCA_TABS.HEATERS);
    fbLakeshoreButton    : FB_HMI_BUTTON(sName := 'Lakeshore'            , sIconName := '', nThisTab := E_HMI_SCA_TABS.LAKESHORE_DET);
    fbTControlButton     : FB_HMI_BUTTON(sName := 'Control loops'        , sIconName := '', nThisTab := E_HMI_SCA_TABS.TCONTROL);
    
    // connection status
    sConnected           : STRING;
    eConnectedColor      : E_HMI_COLORS;
END_VAR

// update the connection status
sConnected      := F_GetConnectionString(bConnected);
eConnectedColor := F_GetConnectionColor(bConnected); 

// update the components
fbTemperatures( fbInstance := temperatures      , bConnected := bConnected);
fbVoters(       fbInstance := voters            , bConnected := bConnected);
fbTControl(     fbInstance := tctrl             , bConnected := bConnected);
fbHeaters(      fbInstance := heaters           , bConnected := bConnected);
fbLakeshore(    fbInstance := lakeshores.ls_sca , bConnected := bConnected);

// update the buttons
// sca
fbTemperaturesButton(
    stColor     := fbTemperatures.fbStatusColor,
    nActiveTab  := eActiveTab,
    sActiveName := sActiveName);
fbVotersButton(
    stColor     := fbVoters.fbStatusColor,
    nActiveTab  := eActiveTab,
    sActiveName := sActiveName);
fbHeatersButton(
    stColor     := fbHeaters.fbStatusColor,
    nActiveTab  := eActiveTab,
    sActiveName := sActiveName);
fbLakeshoreButton(
    stColor     := fbLakeshore.fbStatusColor,
    nActiveTab  := eActiveTab,
    sActiveName := sActiveName);
fbTControlButton(
    stColor     := fbTControl.fbStatusColor,
    nActiveTab  := eActiveTab,
    sActiveName := sActiveName);

// update the summary health/busy status
fbHealthStatus(
    bIsEnabled  := bConnected,
    bIsGood     :=     fbTemperatures.fbHealthStatus.bGood
                   AND fbVoters.fbHealthStatus.bGood
                   AND fbTControl.fbHealthStatus.bGood
                   AND fbHeaters.fbHealthStatus.bGood
                   AND fbLakeshore.fbHealthStatus.bGood,
    bHasWarning :=     fbTemperatures.fbHealthStatus.bWarning
                    OR fbVoters.fbHealthStatus.bWarning
                    OR fbTControl.fbHealthStatus.bWarning
                    OR fbHeaters.fbHealthStatus.bWarning
                    OR fbLakeshore.fbHealthStatus.bWarning);

fbBusyStatus(
    bIsEnabled   := bConnected,
    bIsBusy      :=    fbTemperatures.fbBusyStatus.bBusy
                    OR fbVoters.fbBusyStatus.bBusy
                    OR fbTControl.fbBusyStatus.bBusy
                    OR fbHeaters.fbBusyStatus.bBusy
                    OR fbLakeshore.fbBusyStatus.bBusy);

M_UpdateStatusColor();

END_FUNCTION_BLOCK

// HMI/POUs/Util/FB_HMI_BACK
FUNCTION_BLOCK FB_HMI_BACK EXTENDS FB_HMI_COMPONENT
VAR_INPUT
END_VAR
VAR_OUTPUT
END_VAR
VAR
END_VAR

END_FUNCTION_BLOCK

// HMI/POUs/Util/FB_HMI_CRYO_SIM
FUNCTION_BLOCK FB_HMI_CRYO_SIM EXTENDS FB_HMI_COMPONENT
VAR_INPUT
END_VAR
VAR_OUTPUT
END_VAR
VAR
END_VAR

// update the summary health/busy status
fbHealthStatus(
    bIsEnabled  := TRUE,
    bIsGood     := TRUE);

fbBusyStatus(
    bIsEnabled   := TRUE,
    bIsBusy      := TRUE);

M_UpdateStatusColor();

END_FUNCTION_BLOCK

// HMI/PRG_HMI
{attribute 'OPC.UA.DA' := '0'}
PROGRAM PRG_HMI
VAR
    // System health & busy status
    fbHealthStatus: 		FB_HMI_HEALTH_STATUS;
    fbBusyStatus: 			FB_HMI_BUSY_STATUS;
    fbStatusColor: 			T_HMI_COLORS;
	
	    // active tab of the main frame
    eActiveTab : E_HMI_TABS := E_HMI_TABS.HOME;
    sActiveName : STRING;
	
	ePreviousTab  : E_HMI_TABS := E_HMI_TABS.HOME;
    
    // BUTTONS
    // ===============================================================================================
    
    // buttons at the main screen
    fbHomeButton: 			FB_HMI_BUTTON('Home'     , 		'Start'      , 	E_HMI_TABS.HOME);
    fbServicesButton : 		FB_HMI_BUTTON('Services' , 		'Services'   , 	E_HMI_TABS.SERVICES);	
	fbEventsButton: 		FB_HMI_BUTTON('Events' , 		'Events'     , 	E_HMI_TABS.EVENTS);
	fbIcsInterlocksButton: 	FB_HMI_BUTTON('ICS Interlocks' ,'Interlock'  ,  E_HMI_TABS.ICS_INTERLOCKS);
	fbCryoSimButton: 		FB_HMI_BUTTON('Simulation' ,	'' 			 ,  E_HMI_TABS.SIMULATION);
	
	fbBackButton: 			FB_HMI_BUTTON('Back'     , 		''      	 , 	ePreviousTab);
    
    // Subsystem buttons
    fbCryButton: 	        FB_HMI_BUTTON('CRY'      , ''   , E_HMI_TABS.SUBSYSTEMS_CRY);
    fbCfoButton: 	        FB_HMI_BUTTON('CFO'      , ''   , E_HMI_TABS.SUBSYSTEMS_CFO);
    fbImgButton: 	        FB_HMI_BUTTON('IMG'      , ''   , E_HMI_TABS.SUBSYSTEMS_IMG);
    fbLmsButton: 	        FB_HMI_BUTTON('LMS'      , ''   , E_HMI_TABS.SUBSYSTEMS_LMS);
    fbScaButton: 	        FB_HMI_BUTTON('SCA'      , ''   , E_HMI_TABS.SUBSYSTEMS_SCA);
    fbIcsButton: 	        FB_HMI_BUTTON('ICS'      , ''   , E_HMI_TABS.SUBSYSTEMS_ICS);
	
	// Cryo Routines buttons
	fbEvacuationButton: 	FB_HMI_BUTTON('Evacuation' , 	'', 	E_HMI_TABS.EVACUATION);
	fbCoolDownButton: 		FB_HMI_BUTTON('Cool-Down' , 	'', 	E_HMI_TABS.COOL_DOWN);
	fbWarmUpButton: 		FB_HMI_BUTTON('Warm-Up' , 		'', 		E_HMI_TABS.WARM_UP);
	fbVentingButton: 		FB_HMI_BUTTON('Venting' , 		'', 		E_HMI_TABS.VENTING);
	fbRegenerationButton: 	FB_HMI_BUTTON('Regeneration' , 	'', E_HMI_TABS.REGENERATION);
	fbPowerOutageButton: 	FB_HMI_BUTTON('Power-Outage' , 	'', E_HMI_TABS.POWER_OUTAGE);
	fbAntiFoggingButton: 	FB_HMI_BUTTON('Anti-Fogging' , 	'', E_HMI_TABS.ANTI_FOGGING);
	
	// Cryo devices buttons
	
	fbDevicesButton: 		FB_HMI_BUTTON('Devices' , 		'', 	eActiveTab);
	
	fbCabinetsButton: 		FB_HMI_BUTTON('Cabinets' , 		'', 	E_HMI_TABS.CABINETS);
	fbValvesButton: 		FB_HMI_BUTTON('Valves' , 		'', 	E_HMI_TABS.VALVES);
	fbControlUnitsButton: 	FB_HMI_BUTTON('Control Units' , '',		E_HMI_TABS.CONTROL_UNITS);
	fbHeatersButton: 		FB_HMI_BUTTON('Heaters' , 		'', 	E_HMI_TABS.HEATERS);
	fbPressuresButton: 		FB_HMI_BUTTON('Pressures' , 	'', 	E_HMI_TABS.PRESSURES);
	fbCoolersButton: 		FB_HMI_BUTTON('Coolers' , 		'', 	E_HMI_TABS.COOLERS);
	fbPumpsButton: 			FB_HMI_BUTTON('Pumps' , 		'', 	E_HMI_TABS.PUMPS);
	fbTemperaturesButton: 	FB_HMI_BUTTON('Temperatures' , 	'', 	E_HMI_TABS.TEMPERATURES);
	fbDetectorsButton: 		FB_HMI_BUTTON('Detectors' , 	'', 	E_HMI_TABS.DETECTORS);
	fbControlLoopsButton: 	FB_HMI_BUTTON('Control Loops' , '', 	E_HMI_TABS.CONTROL_LOOPS);
	
    // COMPONENTS
    // ===============================================================================================
    
    // general
    fbServices: 			FB_HMI_SERVICES;
	fbEvents: 				FB_HMI_EVENTS;
	fbIcsInterlocks: 		FB_HMI_ICS_INTERLOCKS;
	fbCryoSim: 				FB_HMI_CRYO_SIM;
	
	fbBack: 				FB_HMI_BACK;
	
	// Cryo Routines
	fbEvacuation: 			FB_HMI_EVACUATION;
	fbCoolDown: 			FB_HMI_COOL_DOWN;	
	fbWarmUp: 				FB_HMI_WARM_UP;
	fbVenting: 				FB_HMI_VENTING;
	fbRegeneration: 		FB_HMI_REGENERATION;
	fbPowerOutage: 			FB_HMI_POWER_OUTAGE;
	fbAntiFogging: 			FB_HMI_ANTI_FOGGING;
	
	// Cryo devices status
	
	fbDevices: 				FB_HMI_DEVICES;
	
	fbCabinets: 			FB_HMI_CABINETS;
	fbValves: 				FB_HMI_VALVES;
	fbControlUnits: 		FB_HMI_CONTROL_UNITS;
	fbHeaters: 				FB_HMI_HEATERS;
	fbPressures: 			FB_HMI_PRESSURES;
	fbCoolers: 				FB_HMI_COOLERS;
	fbPumps: 				FB_HMI_PUMPS;
	fbTemperatures: 		FB_HMI_TEMPERATURES;
    fbDetectors: 			FB_HMI_DETECTORS;
	fbControlLoops:			FB_HMI_CONTROL_LOOPS;
	
    // subsystems
    {attribute 'OPC.UA.DA' := '0'}
    fbCry:                  FB_HMI_CRY;
    {attribute 'OPC.UA.DA' := '0'}
    fbCfo:                  FB_HMI_CFO;
    {attribute 'OPC.UA.DA' := '0'}
    fbImg:                  FB_HMI_IMG;
    {attribute 'OPC.UA.DA' := '0'}
    fbLms:                  FB_HMI_LMS;
    {attribute 'OPC.UA.DA' := '0'}
    fbSca:                  FB_HMI_SCA;
    {attribute 'OPC.UA.DA' := '0'}
    fbIcs:                  FB_HMI_ICS;
    

    // Internal persistent state (survives method calls)
    _eLastTab       : E_HMI_TABS := E_HMI_TABS.HOME;
    _bInitDone      : BOOL := FALSE;
END_VAR

M_TrackPreviousTab(
    eActiveTabIn := eActiveTab,
    ePreviousTabOut => ePreviousTab,
    bTabChanged => 
);

//// update the components
fbServices(fbInstance := MAIN.fbServices);
fbEvents(); 				
fbIcsInterlocks();
fbCryoSim();

fbBack(); 		

// Cryo Routines
fbEvacuation(fbInstance := MAIN.met_cryo_ctrl.met_evac, interlocks := MAIN.met_cryo_ctrl.interlocks);			
fbCoolDown(fbInstance := MAIN.met_cryo_ctrl.met_cool_down, interlocks := MAIN.met_cryo_ctrl.interlocks);	
fbWarmUp(fbInstance := MAIN.met_cryo_ctrl.met_warm_up, interlocks := MAIN.met_cryo_ctrl.interlocks);			
fbVenting(fbInstance := MAIN.met_cryo_ctrl.met_venting, interlocks := MAIN.met_cryo_ctrl.interlocks); 				
fbRegeneration(fbInstance := MAIN.met_cryo_ctrl.met_regeneration, interlocks := MAIN.met_cryo_ctrl.interlocks); 		
fbPowerOutage();
fbAntiFogging(fbInstance := MAIN.met_cryo_ctrl.met_anti_fogging, interlocks := MAIN.met_cryo_ctrl.interlocks);			

// Cryo devices status
fbCabinets(); 			
fbValves(); 				
fbControlUnits(); 		
fbHeaters();				
fbPressures(); 			
fbCoolers(); 				
fbPumps();			
fbTemperatures(voters       := MAIN.met_cryo_ctrl.met_voters); 		
fbDetectors();
fbControlLoops();

// Subsystems
fbCry(
    temperatures := MAIN.met_cryo_ctrl.met_temp,
    rh           := MAIN.met_cryo_ctrl.met_rh,
    heaters      := MAIN.met_cryo_ctrl.met_heaters,
    voters       := MAIN.met_cryo_ctrl.met_voters,
    tctrl        := MAIN.met_cryo_ctrl.met_tctrl,
	ln2ctrl      := MAIN.met_cryo_ctrl.met_cool_down.lc_ln2_level_ctrl);
fbCfo(
    temperatures := MAIN.met_cryo_ctrl.met_temp,
    heaters      := MAIN.met_cryo_ctrl.met_heaters,
    voters       := MAIN.met_cryo_ctrl.met_voters,
    tctrl        := MAIN.met_cryo_ctrl.met_tctrl);
fbImg(
    bConnected   := TRUE,
    temperatures := MAIN.met_cryo_ctrl.met_temp,
    heaters      := MAIN.met_cryo_ctrl.met_heaters,
    voters       := MAIN.met_cryo_ctrl.met_voters,
    tctrl        := MAIN.met_cryo_ctrl.met_tctrl,
    lakeshores   := MAIN.met_cryo_ctrl.met_lakeshores);
fbSca(
    bConnected   := TRUE,
    temperatures := MAIN.met_cryo_ctrl.met_temp,
    heaters      := MAIN.met_cryo_ctrl.met_heaters,
    voters       := MAIN.met_cryo_ctrl.met_voters,
    tctrl        := MAIN.met_cryo_ctrl.met_tctrl,
    lakeshores   := MAIN.met_cryo_ctrl.met_lakeshores);
fbLms(
    temperatures := MAIN.met_cryo_ctrl.met_temp,
    heaters      := MAIN.met_cryo_ctrl.met_heaters,
    voters       := MAIN.met_cryo_ctrl.met_voters,
    tctrl        := MAIN.met_cryo_ctrl.met_tctrl);
fbIcs(
    ccus         := MAIN.met_cryo_ctrl.met_ccus);


// update the status
M_UpdateStatus();

// update the system-level buttons
fbHomeButton(stColor := fbStatusColor, nActiveTab := eActiveTab, sActiveName := sActiveName);
// buttons at the main screen 
fbServicesButton(stColor := fbServices.fbStatusColor, nActiveTab := eActiveTab, sActiveName := sActiveName);	
fbEventsButton(stColor:= fbEvents.fbStatusColor, nActiveTab:= eActiveTab, sActiveName:= sActiveName);		
fbIcsInterlocksButton(stColor:= fbIcsInterlocks.fbStatusColor, nActiveTab:= eActiveTab, sActiveName:= sActiveName); 	

// Simulation Button

fbCryoSimButton(stColor:= fbCryoSim.fbStatusColor, nActiveTab:= eActiveTab, sActiveName:= sActiveName);

// Cryo Routines
fbEvacuationButton(stColor:= fbEvacuation.fbStatusColor, nActiveTab:= eActiveTab, sActiveName:= sActiveName); 	
fbCoolDownButton(stColor:= fbCoolDown.fbStatusColor, nActiveTab:= eActiveTab, sActiveName:= sActiveName); 		
fbWarmUpButton(stColor:= fbWarmUp.fbStatusColor, nActiveTab:= eActiveTab, sActiveName:= sActiveName); 		

fbVentingButton(stColor:= fbVenting.fbStatusColor, nActiveTab:= eActiveTab, sActiveName:= sActiveName); 		

fbRegenerationButton(stColor:= fbRegeneration.fbStatusColor, nActiveTab:= eActiveTab, sActiveName:= sActiveName);	
fbPowerOutageButton(stColor:= fbPowerOutage.fbStatusColor, nActiveTab:= eActiveTab, sActiveName:= sActiveName);
fbAntiFoggingButton(stColor:= fbAntiFogging.fbStatusColor, nActiveTab:= eActiveTab, sActiveName:= sActiveName); 	

// Cryo devices status

fbDevicesButton(stColor:= fbDevices.fbStatusColor, nActiveTab:= eActiveTab, sActiveName:= sActiveName); 

fbBackButton(stColor:= fbBack.fbStatusColor, nActiveTab:= ePreviousTab, sActiveName:= sActiveName); 

fbCabinetsButton(stColor:= fbCabinets.fbStatusColor, nActiveTab:= eActiveTab, sActiveName:= sActiveName); 		
fbValvesButton(stColor:= fbValves.fbStatusColor, nActiveTab:= eActiveTab, sActiveName:= sActiveName); 		
fbControlUnitsButton(stColor:= fbControlUnits.fbStatusColor, nActiveTab:= eActiveTab, sActiveName:= sActiveName);	
fbHeatersButton(stColor:= fbHeaters.fbStatusColor, nActiveTab:= eActiveTab, sActiveName:= sActiveName); 		
fbPressuresButton(stColor:= fbPressures.fbStatusColor, nActiveTab:= eActiveTab, sActiveName:= sActiveName); 		
fbCoolersButton(stColor:= fbCoolers.fbStatusColor, nActiveTab:= eActiveTab, sActiveName:= sActiveName); 		
fbPumpsButton(stColor:= fbPumps.fbStatusColor, nActiveTab:= eActiveTab, sActiveName:= sActiveName); 			
fbTemperaturesButton(stColor:= fbTemperatures.fbStatusColor, nActiveTab:= eActiveTab, sActiveName:= sActiveName); 	
fbDetectorsButton(stColor:= fbDetectors.fbStatusColor, nActiveTab:= eActiveTab, sActiveName:= sActiveName);
fbControlLoopsButton(stColor:= fbControlLoops.fbStatusColor, nActiveTab:= eActiveTab, sActiveName:= sActiveName);

// Subsystem buttons
fbCryButton(stColor:= fbCry.fbStatusColor, nActiveTab:= eActiveTab, sActiveName:= sActiveName);
fbCfoButton(stColor:= fbCfo.fbStatusColor, nActiveTab:= eActiveTab, sActiveName:= sActiveName);
fbImgButton(stColor:= fbImg.fbStatusColor, nActiveTab:= eActiveTab, sActiveName:= sActiveName);
fbLmsButton(stColor:= fbLms.fbStatusColor, nActiveTab:= eActiveTab, sActiveName:= sActiveName);
fbScaButton(stColor:= fbSca.fbStatusColor, nActiveTab:= eActiveTab, sActiveName:= sActiveName);
fbIcsButton(stColor:= fbIcs.fbStatusColor, nActiveTab:= eActiveTab, sActiveName:= sActiveName);

METHOD M_TrackPreviousTab : BOOL
VAR_INPUT
    eActiveTabIn : E_HMI_TABS;
END_VAR
VAR_OUTPUT
    ePreviousTabOut : E_HMI_TABS;
    bTabChanged     : BOOL;
END_VAR
// One-time initialization
IF NOT _bInitDone THEN
    _eLastTab       := eActiveTabIn;
    ePreviousTabOut := eActiveTabIn; // no previous yet; define as current
    bTabChanged     := FALSE;
    _bInitDone      := TRUE;
ELSE
    bTabChanged := (eActiveTabIn <> _eLastTab);
    IF bTabChanged THEN
        ePreviousTabOut := _eLastTab;   // report the previous
        _eLastTab       := eActiveTabIn; // store new current for next time
    ELSE
        // keep the last known previous in the FB variable if you mirror it outside
        ePreviousTabOut := ePreviousTab; // or keep last output value
    END_IF
END_IF
END_METHOD

METHOD M_UpdateStatus
VAR_INPUT
END_VAR
// update the health & busy statuses
//fbHealthStatus(
//    bIsEnabled :=   fbImg.fbHealthStatus.bEnabled
//                AND fbSca.fbHealthStatus.bEnabled,
//    bIsGood :=      fbImg.fbHealthStatus.bGood
//                AND fbSca.fbHealthStatus.bGood);
              //AND fbServices.fbHealthStatus.bGood
              //AND fbLms.fbHealthStatus.bGood (* AND ... *));
//fbBusyStatus(
//    bIsEnabled :=   fbImg.fbBusyStatus.bEnabled
//                AND fbSca.fbBusyStatus.bEnabled,
//    bIsBusy := fbServices.fbBusyStatus.bBusy 
//                 OR fbImg.fbBusyStatus.bBusy 
//                 OR fbLms.fbBusyStatus.bBusy 
//                 OR fbSca.fbBusyStatus.bBusy);

fbStatusColor := F_HMI_HEALTH_BUSY_TO_COLOR(fbHealthStatus, fbBusyStatus);
END_METHOD

END_PROGRAM

// POUs/Devices/Heaters/Heater_Ctrl/FB_HEATER_CPAU60
FUNCTION_BLOCK FB_HEATER_CPAU60
VAR_INPUT
	{attribute 'OPC.UA.DA' := '0'}	
	in_sName:						STRING 	:= 'Heater Controller CXWUI60';	// Controller name	
	{attribute 'OPC.UA.DA' := '0'}
	in_nHeaterResistance:			INT;			// Resistance of the heater to be controlled [Ohms]
	{attribute 'OPC.UA.DA' := '0'}
	in_nMaxHeaterPower:				INT;			// Max power of the heater to be controlled [Ohms]
	
END_VAR
VAR
	{attribute 'OPC.UA.DA' := '0'}
	i_nCouplerState		AT%I*:		UINT;		// Terminal state. Should be 8, i.e. OP.
	{attribute 'OPC.UA.DA' := '0'}
	q_bEnable			AT%Q*:		BOOL;		// Enable heater power
	{attribute 'OPC.UA.DA' := '0'}
	q_nSetVoltage		AT%Q*:		INT := 0;	// Adjustable PS voltage [0 - 16383 (0 - 5V)] for liner power supply to power the heater
	
 	{attribute 'OPC.UA.DA' := '0'}
	i_nActCurrent		AT%I*:		DINT;		// Terminal state. Should be 8, i.e. OP.
	{attribute 'OPC.UA.DA' := '0'}
	i_nStatus			AT%I*:		UINT;		// EL3164 input status (might implement if needed)

	stat:		T_METIS_CRYO_HEATER_STATUS;
	ctrl:		T_METIS_CRYO_HEATER_CTRL;

	lrGetPowerVar:		LREAL;	
	bManualInputFlag:			BOOL := TRUE;
	lrManualHeaterPower:		LREAL := 1.7; // random init value
	
	
END_VAR



IF ctrl.bEnable THEN
	q_bEnable := TRUE;
	stat.bActive := TRUE;
ELSE
	q_bEnable := FALSE;
	stat.bActive := FALSE;
END_IF

//M_Configure();

M_ReadInputs();

M_SetStatus();

M_SetCtrlOutput();

PROPERTY bIsActive : BOOL
GET
bIsActive := stat.bActive;
END_GET
END_PROPERTY

PROPERTY bIsInError : BOOL
GET
bIsInError := stat.bError;
END_GET
END_PROPERTY

PROPERTY bIsNotActive : BOOL
GET
bIsNotActive := NOT stat.bActive;
END_GET
END_PROPERTY

PROPERTY lrHeaterPower : LREAL
GET
lrHeaterPower := ctrl.lrPower;
END_GET
SET
ctrl.lrPower := lrHeaterPower;
END_SET
END_PROPERTY

METHOD M_Activate
VAR_INPUT
END_VAR
ctrl.bEnable := TRUE;
END_METHOD

METHOD M_Configure : BOOL
VAR_INPUT
END_VAR


//ctrl.lrPower := in_lrHeaterPower;
END_METHOD

METHOD M_DeActivate
VAR_INPUT
END_VAR
ctrl.bEnable := FALSE;
END_METHOD

METHOD M_GetHeaterPower : BOOL
VAR_INPUT
	m_lrHeaterPower:  LREAL;
END_VAR
//lrManualHeaterPower := m_lrHeaterPower;

lrGetPowerVar := m_lrHeaterPower;
END_METHOD

METHOD M_ReadInputs
VAR_INPUT
END_VAR
VAR
	m_nActCurrent:		DINT;
END_VAR
(*
	Read all inputs and assign values to variables.
*)

m_nActCurrent	:=	i_nActCurrent;

M_ScaleInput(m_nActCurrent:= m_nActCurrent);
END_METHOD

METHOD M_ScaleInput : BOOL
VAR_INPUT
	m_nActCurrent:	DINT;
END_VAR

(*EL3681 Digital Multimeter terminal

Scaled presentation:
corresponds to 1 bit per µV / µA,
Examples:
Mode 0, Autorange, 2.5 V: 2,500,000 decimal
Mode 2, 800 mA: 800,000 decimal

  *) 
stat.lrActCurrent :=  DINT_TO_LREAL(m_nActCurrent) / 1000000.0;
END_METHOD

METHOD M_ScaleOutput : BOOL
VAR_INPUT
	m_lrCtrlCurrent	:	LREAL;
	m_lrCtrlVoltage	:   LREAL;
END_VAR



//Set voltage
// AI from terminal is type INT. Full scale reading (0 - 32767) represent 0 to 10V. 
// We read 0 - 10V, so we scale from 0 t 32767 => 10/32767 =  0.00030518509
// Max Output voltage at 16383 is 60. First translate 0 - 60 into 0 - 10 (10/60 = 0.166666 ) then 0 - 10 to 0 to 32767


q_nSetVoltage := LREAL_TO_INT( (m_lrCtrlVoltage * 0.166666) / 0.00030518509);
END_METHOD

METHOD M_SetCtrlOutput : BOOL
VAR
	m_lrCtrlPower 	: 	LREAL;
	m_lrCtrlCurrent	:	LREAL;
	m_lrCtrlVoltage	:	LREAL;	 
END_VAR


////Enable the heater
//q_bEnable := ctrl.bEnable;

// Scale power value

m_lrCtrlPower := 	(ctrl.lrPower/100)*in_nMaxHeaterPower;
//m_lrCtrlPower := 	(in_lrHeaterPower/100)*in_nMaxHeaterPower;


m_lrCtrlCurrent	:=  SQRT(m_lrCtrlPower/in_nHeaterResistance);

m_lrCtrlVoltage	:=	SQRT(m_lrCtrlPower * in_nHeaterResistance); 


M_ScaleOutput(m_lrCtrlCurrent := m_lrCtrlCurrent, m_lrCtrlVoltage := m_lrCtrlVoltage);
END_METHOD

METHOD M_SetHeaterPower : LREAL
VAR_INPUT
END_VAR
M_SetHeaterPower := lrGetPowerVar;
END_METHOD

METHOD M_SetManualInputFlag : BOOL
VAR_INPUT
	m_bManual_Input_Flag:		BOOL;
END_VAR
bManualInputFlag := m_bManual_Input_Flag;
END_METHOD

METHOD M_SetStatus : BOOL
VAR_INPUT
END_VAR

// Set actual power I^2R
stat.lrActHeaterPower := stat.lrActCurrent * stat.lrActCurrent * in_nHeaterResistance;

// Set max current
IF in_nHeaterResistance > 0 THEN
stat.lrMaxCurrent :=  SQRT(INT_TO_REAL(in_nMaxHeaterPower)/INT_TO_REAL(in_nHeaterResistance));
ELSE
	stat.lrMaxCurrent := 999.9;
END_IF

//IF ctrl.bEnable = TRUE THEN
//	stat.bActive := TRUE;
//ELSE
//	stat.bActive := FALSE;
//END_IF


stat.bHeaterOpenLoop := (stat.lrActCurrent <= 0)
                        AND stat.bActive 
                        AND (ctrl.lrPower > 0);
 
// Check if there is a short circuit: Comparing the actual current with the Max current + 1 A  
 IF stat.lrActCurrent > (stat.lrMaxCurrent + 1) THEN
	 stat.bHeaterShort := TRUE;
 ELSE
	stat.bHeaterShort := FALSE;
 END_IF
END_METHOD

END_FUNCTION_BLOCK

// POUs/Devices/Heaters/Heater_Ctrl/FB_HEATER_CXWUI60
FUNCTION_BLOCK FB_HEATER_CXWUI60
VAR_INPUT
	{attribute 'OPC.UA.DA' := '0'}	
	in_sName:						STRING := 'Heater Controller CXWUI60';	// Controller name
	{attribute 'OPC.UA.DA' := '0'}
	in_nHeaterResistance:			INT;			// Resistance of the heater to be controlled [Ohms]
	{attribute 'OPC.UA.DA' := '0'}
	in_nMaxHeaterPower:			INT;			// Max power of the heater to be controlled [Ohms]
	
END_VAR
VAR
	{attribute 'OPC.UA.DA' := '0'}
	i_nCouplerState		AT%I*:		UINT;		// Terminal state. Should be 8, i.e. OP.
	{attribute 'OPC.UA.DA' := '0'}
	q_bEnable			AT%Q*:		BOOL;		// Enable heater power
	{attribute 'OPC.UA.DA' := '0'}
	q_nSetVoltage		AT%Q*:		INT := 0;	// Adjustable PS voltage [0 - 16383 (0 - 5V)] for liner power supply to power the heater
	{attribute 'OPC.UA.DA' := '0'}
	q_nSetCurrent		AT%Q*:		INT := 0;	// Adjustable PS current [0 - 16383 (0 - 4Amps)] for liner power supply to power the heater
 	{attribute 'OPC.UA.DA' := '0'}
	i_nActCurrent		AT%I*:		INT;		// Terminal state. Should be 8, i.e. OP.
	{attribute 'OPC.UA.DA' := '0'}
	i_nStatus			AT%I*:		UINT;		// EL3164 input status (might implement if needed)

	stat:		T_METIS_CRYO_HEATER_STATUS;
	ctrl:		T_METIS_CRYO_HEATER_CTRL;

	lrGetPowerVar:		LREAL;
	bManualInputFlag:			BOOL := TRUE;
	lrManualHeaterPower:		LREAL := 1.7; // random init value
	
END_VAR



IF ctrl.bEnable THEN
	q_bEnable := TRUE;
	stat.bActive := TRUE;
ELSE
	q_bEnable := FALSE;
	stat.bActive := FALSE;
END_IF

//M_Configure();

M_ReadInputs();

M_SetStatus();

M_SetCtrlOutput();

PROPERTY bIsActive : BOOL
GET
bIsActive := stat.bActive;
END_GET
END_PROPERTY

PROPERTY bIsInError : BOOL
GET
bIsInError := stat.bError;
END_GET
END_PROPERTY

PROPERTY bIsNotActive : BOOL
GET
bIsNotActive := NOT stat.bActive;
END_GET
END_PROPERTY

PROPERTY lrHeaterPower : LREAL
GET
lrHeaterPower := ctrl.lrPower;
END_GET
SET
ctrl.lrPower := lrHeaterPower;
END_SET
END_PROPERTY

METHOD M_Activate
VAR_INPUT
END_VAR
ctrl.bEnable := TRUE;
END_METHOD

METHOD M_Configure : BOOL
VAR_INPUT
END_VAR


//ctrl.lrPower := in_lrHeaterPower;
END_METHOD

METHOD M_DeActivate
VAR_INPUT
END_VAR
ctrl.bEnable := FALSE;
END_METHOD

METHOD M_GetHeaterPower : BOOL
VAR_INPUT
	m_lrHeaterPower:  LREAL;
END_VAR
//lrManualHeaterPower := m_lrHeaterPower;

lrGetPowerVar := m_lrHeaterPower;
END_METHOD

METHOD M_ReadInputs
VAR_INPUT
END_VAR
VAR
	m_nActCurrent:		INT;
END_VAR
(*
	Read all inputs and assign values to variables.
*)

m_nActCurrent	:=	i_nActCurrent;

M_ScaleInput(m_nActCurrent:= m_nActCurrent);
END_METHOD

METHOD M_ScaleInput : BOOL
VAR_INPUT
	m_nActCurrent:	INT;
END_VAR


// AI from terminal is type INT. Full scale reading (0 - 32767) represent 0 to 10V. 
// We read only 0 - 5V, so we scale from 0 t 16383 => 5/16383 = 0.0003051944
   
stat.lrActCurrent :=  m_nActCurrent * 0.0003051944;
END_METHOD

METHOD M_ScaleOutput : BOOL
VAR_INPUT
	m_lrCtrlCurrent	:	LREAL;
	m_lrCtrlVoltage	:   LREAL;
END_VAR




//Set current 
q_nSetCurrent := LREAL_TO_INT(m_lrCtrlCurrent / 0.0003051944);

//Set voltage
// AI from terminal is type INT. Full scale reading (0 - 32767) represent 0 to 10V. 
// We read only 0 - 5V, so we scale from 0 t 16383 => 5/16383 = 0.0003051944
// Max Output voltage at 16383 is 60. First translate 0 - 60 into 0 - 5 (5/60 = 0.08333) then 0 - 5 to 0 to 16383


q_nSetVoltage := LREAL_TO_INT( (m_lrCtrlVoltage * 0.08333) / 0.0003051944 );
END_METHOD

METHOD M_SetCtrlOutput : BOOL
VAR
	m_lrCtrlPower 	: 	LREAL;
	m_lrCtrlCurrent	:	LREAL;
	m_lrCtrlVoltage	:	LREAL;	 
END_VAR


////Enable the heater
//q_bEnable := ctrl.bEnable;

// Scale power value

m_lrCtrlPower := 	(ctrl.lrPower/100)*in_nMaxHeaterPower;
//m_lrCtrlPower := 	(in_lrHeaterPower/100)*in_nMaxHeaterPower;


m_lrCtrlCurrent	:=  SQRT(m_lrCtrlPower/in_nHeaterResistance);

m_lrCtrlVoltage	:=	SQRT(m_lrCtrlPower * in_nHeaterResistance); 


M_ScaleOutput(m_lrCtrlCurrent := m_lrCtrlCurrent, m_lrCtrlVoltage := m_lrCtrlVoltage);
END_METHOD

METHOD M_SetHeaterPower : LREAL
VAR_INPUT
END_VAR
M_SetHeaterPower := lrGetPowerVar;
END_METHOD

METHOD M_SetManualInputFlag : BOOL
VAR_INPUT
	m_bManual_Input_Flag:		BOOL;
END_VAR
bManualInputFlag := m_bManual_Input_Flag;
END_METHOD

METHOD M_SetStatus : BOOL
VAR_INPUT
END_VAR

// Set actual power I^2R
stat.lrActHeaterPower := stat.lrActCurrent * stat.lrActCurrent * in_nHeaterResistance;

// Set max current
IF in_nHeaterResistance > 0 THEN
stat.lrMaxCurrent :=  SQRT(INT_TO_REAL(in_nMaxHeaterPower)/INT_TO_REAL(in_nHeaterResistance));
ELSE
	stat.lrMaxCurrent := 999.9;
END_IF

//IF ctrl.bEnable = TRUE THEN
//	stat.bActive := TRUE;
//ELSE
//	stat.bActive := FALSE;
//END_IF


 IF stat.lrActCurrent <= 0 THEN
	 stat.bHeaterOpenLoop := TRUE;
 ELSE
	stat.bHeaterOpenLoop := FALSE;
 END_IF

 
// Check if there is a short circuit: Comparing the actual current with the Max current + 1 A  
 IF stat.lrActCurrent > (stat.lrMaxCurrent + 1) THEN
	 stat.bHeaterShort := TRUE;
 ELSE
	stat.bHeaterShort := FALSE;
 END_IF
END_METHOD

END_FUNCTION_BLOCK

// POUs/Devices/Temp_Voter/FB_METIS_VOTER_COPY_for_new_HMI
{attribute 'TcHmiSymbol.Show'}
FUNCTION_BLOCK FB_METIS_VOTER_COPY_for_new_HMI
VAR_INPUT
	{attribute 'OPC.UA.DA' := '0'}
	in_sName:	STRING;
	{attribute 'OPC.UA.DA' := '0'}
	in_bSimulation:	BOOL	:= FALSE;	// If TRUE, the temperature value is simulated.
	{attribute 'OPC.UA.DA' := '0'}
	in_nRampPeriodSec:		UDINT := 60;	// Ramp measurement period [sec]. Default 60 sec.
END_VAR
VAR_IN_OUT
	{attribute 'OPC.UA.DA' := '0'}
	met_temp: FB_METIS_TEMPERATURES;
	
END_VAR
VAR
(****** Keeping this for PLC Visus ****)	
	{attribute 'OPC.UA.DA' := '0'}
	aTempIndexes:		ARRAY[0..4] OF INT;
	{attribute 'OPC.UA.DA' := '0'}
	nVoteMethod:		E_METIS_TEMP_VOTE_METHOD;
    (* Enabled or disabled *)
    bEnabled:       BOOL;
(**************************************)	

	cfg:				T_METIS_TEMP_VOTE_CFG;

	{attribute 'OPC.UA.DA' := '0'}
	aTempPointers:	    ARRAY[0..4] OF POINTER TO FB_METIS_TEMPERATURE;
// 	{attribute 'OPC.UA.DA' := '0'}
// 	aTempIndexes:		ARRAY[0..4] OF INT := [0, 0, 0, 0, 0];


	{attribute 'TcHmiSymbol.Show'}
	{attribute 'OPC.UA.DA' := '1'}
	{attribute 'OPC.UA.DA.Access' := '1'}
	stat	: T_METIS_CRYO_TEMP_VOTE_STATUS;
    

    
    (* User description *)
    sDescription:   STRING;
    
	(*Engineering MODE*)
	bEngMode:		BOOL := FALSE;
	bAutoMode:		BOOL := TRUE;
	bManualMode:	BOOL := FALSE;	

	(*Configuration*)
	bConfigured:	BOOL := FALSE;
	
	(*Read/Write configuration*)
	{attribute 'OPC.UA.DA' := '0'}
	fbTempVoteConfig:		FB_READ_WRITE_TEMP_VOTE_CONFIG;
	bReadConfig:			BOOL;
	bWriteConfig:			BOOL;
	(*Ramp *)
	{attribute 'OPC.UA.DA' := '0'}
	bRampTimerStarted:	BOOL := FALSE;
	{attribute 'OPC.UA.DA' := '0'}
	rampTimer:	TON;		// Timer for calculating ramp
	
    // outputs that can be used for linking
	{attribute 'OPC.UA.DA' := '0'}
    q_lrTemp    AT %Q*: LREAL;
	{attribute 'OPC.UA.DA' := '0'}
	q_bToggle   AT %Q*: BOOL;
	{attribute 'OPC.UA.DA' := '0'}
	q_bValid   AT %Q*: BOOL := FALSE;
	
		// Alarm handling
	// List of alarms to be handled by Temperature
	arrEventEntry : ARRAY [0..2] OF TcEventEntry;
	// Alarm handler FB
	fbAlarmHandler : FB_AlarmHandler;
	
	// Logs logs
	logs:	FB_CRYO_FUNCTION_LOG;
	
END_VAR

// to avoid any problem of invalid pointers, set them right away
M_UpdateTempPointers(met_temp := met_temp);

(*Read/Write configuration*)
fbTempVoteConfig(in_sTVoteName:= in_sName, Temp_Vote_Config:= cfg);

IF NOT bConfigured THEN
    M_Configure(met_temp := met_temp);
    RETURN;
END_IF

// set AUTO / MAN / ENG
M_SetPermissionMode();

// read/write the config (if needed)
M_Read_Write_Config(met_temp := met_temp);

M_GetRamp();

M_SetStatus();

PROPERTY bTempNotValid : BOOL
GET
bTempNotValid := NOT stat.bValid;
END_GET
END_PROPERTY

PROPERTY bTempValid : BOOL
GET
bTempValid := stat.bValid;
END_GET
END_PROPERTY

PROPERTY lrRamp : LREAL
GET
lrRamp := stat.lrRamp;
END_GET
END_PROPERTY

PROPERTY lrTempK : LREAL
GET
lrTempK := stat.lrTempK;
END_GET
END_PROPERTY

METHOD M_ConfigReadingFinished
VAR_INPUT
    bError : BOOL;
END_VAR
VAR_IN_OUT
    met_temp : FB_METIS_TEMPERATURES;
END_VAR
VAR
    i : INT;
	sNameString:	STRING; // temp text String 
END_VAR
IF bError THEN
   // ERROR! Just put the indexes to 0
   FOR i := 0 TO 4 DO
       stat.aTempIndexes[i] := 0;
   END_FOR
   stat.bEnabled := FALSE;
   sDescription := in_sName;
ELSE
    // success!
    sNameString := cfg.sTemp1_Name;
    sNameString := cfg.sTemp2_Name;
    sNameString := cfg.sTemp3_Name;
    sNameString := cfg.sTemp4_Name;
    sNameString := cfg.sTemp5_Name;
	stat.aTempIndexes[0] := cfg.eTemperature1;
	stat.aTempIndexes[1] := cfg.eTemperature2;
    stat.aTempIndexes[2] := cfg.eTemperature3;
	stat.aTempIndexes[3] := cfg.eTemperature4;
    stat.aTempIndexes[4] := cfg.eTemperature5;
    stat.nVoteMethod     := cfg.nVote_Method;
    stat.bEnabled        := cfg.bEnabled;
    sDescription    := cfg.sDescription; 
END_IF

M_UpdateTempPointers(met_temp := met_temp);

// clear the flag
fbTempVoteConfig.M_ClearReadingDoneFlag();
END_METHOD

METHOD M_Configure : BOOL
VAR_INPUT
END_VAR
VAR_INST
	{attribute 'OPC.UA.DA' := '0'}
    nConfigureState : INT;
END_VAR
VAR_IN_OUT
	{attribute 'OPC.UA.DA' := '0'}
    met_temp : FB_METIS_TEMPERATURES;
END_VAR
VAR
    i : INT;
END_VAR

CASE nConfigureState OF
    0:  
        // use the name of the voter as the default description
        sDescription := in_sName;
        // start reading the config
        fbTempVoteConfig.M_ReadConfiguration();
        nConfigureState := 1;
    1:
        IF fbTempVoteConfig.bReadingDoneFlag THEN
            M_ConfigReadingFinished(
                bError   := fbTempVoteConfig.bReadError,
                met_temp := met_temp);
            
            bConfigured := TRUE;
        END_IF
END_CASE
END_METHOD

METHOD M_GetRamp
VAR_INPUT
END_VAR
VAR_INST
	{attribute 'OPC.UA.DA' := '0'}
	lrRampStartTempK:	LREAL;	// Temperature at start of ramp timer [K]
END_VAR
VAR
	nRampPeriodSec:		UDINT;	// Ramp measurement period [sec].
END_VAR

IF NOT (stat.bEnabled AND stat.bValid) THEN
    bRampTimerStarted := FALSE;
    stat.lrRamp := 0.0;
    RETURN;
END_IF

IF NOT bRampTimerStarted THEN
	bRampTimerStarted	:= TRUE;
	lrRampStartTempK	:= stat.lrTempK;
	rampTimer(IN:=FALSE);
END_IF

// Execute timer.
// Ramp measurement period should be > 0
nRampPeriodSec	:= in_nRampPeriodSec;
IF nRampPeriodSec = 0 THEN
	nRampPeriodSec	:= 60;
END_IF
rampTimer(IN:=TRUE,PT:=UDINT_TO_TIME(nRampPeriodSec)*1000);

// Calculate ramp at time expiry
IF rampTimer.Q THEN
	// Calculate the temperature ramp per minute
//	IF stat.bValid THEN
		stat.lrRamp	:= (stat.lrTempK - lrRampStartTempK) * 60.0 / nRampPeriodSec;
//	ELSE
//		stat.lrRamp	:= 0.0;
//	END_IF

	// Current temperature is the starting value of the ramp
	lrRampStartTempK	:= stat.lrTempK;

	// Restart the timer
	rampTimer(IN:=FALSE);
END_IF
END_METHOD

METHOD M_Read_Write_Config
VAR_INPUT
END_VAR
VAR_IN_OUT
    met_temp : FB_METIS_TEMPERATURES;
END_VAR
IF bEngMode THEN
    IF bWriteConfig THEN
        
        // update the cfg object
        cfg.bEnabled     := stat.bEnabled;
        cfg.sDescription := sDescription;
        cfg.sTemp1_Name  := aTempPointers[0]^.in_sName;
        cfg.sTemp2_Name  := aTempPointers[1]^.in_sName; 
        cfg.sTemp3_Name  := aTempPointers[2]^.in_sName; 
        cfg.sTemp4_Name  := aTempPointers[3]^.in_sName; 
        cfg.sTemp5_Name  := aTempPointers[4]^.in_sName;
        cfg.nVote_Method := stat.nVoteMethod;
		cfg.eTemperature1:= stat.aTempIndexes[0];
		cfg.eTemperature2:= stat.aTempIndexes[1];
		cfg.eTemperature3:= stat.aTempIndexes[2];
		cfg.eTemperature4:= stat.aTempIndexes[3];
		cfg.eTemperature5:= stat.aTempIndexes[4];
        
        // write the cfg object
        fbTempVoteConfig.M_WriteConfiguration();
        bWriteConfig := FALSE;
                
    ELSIF bReadConfig THEN
	
        fbTempVoteConfig.M_ReadConfiguration();
        bReadConfig := FALSE;

    END_IF
		
END_IF

IF fbTempVoteConfig.bReadingDoneFlag THEN
	M_ConfigReadingFinished(
        bError := fbTempVoteConfig.bReadError,
        met_temp := met_temp);
END_IF
END_METHOD

METHOD M_SetPermissionMode : BOOL
VAR_INPUT
END_VAR
IF bAutoMode THEN
    stat.sStatus    := 'AUTO';
    bManualMode     := FALSE;
    bEngMode        := FALSE;
ELSIF bEngMode	THEN
    stat.sStatus    := 'ENG';
    bManualMode     := FALSE;
    bAutoMode       := FALSE;
ELSIF bManualMode THEN
    stat.sStatus    := 'MANUAL';
    bAutoMode       := FALSE;
    bEngMode        := FALSE;
END_IF
END_METHOD

// Calculate pressure based on the status of the two sensors
METHOD M_SetStatus
VAR_INPUT
END_VAR
VAR
	lrTmp:		LREAL;	// Temporary var
	nSample:	INT;
	i:			INT;
END_VAR
VAR_INST
	{attribute 'OPC.UA.DA' := '0'}
    toggleTimer : TON;
END_VAR
stat.lrSens1TempK := aTempPointers[0]^.stat.lrTempK;
stat.lrSens2TempK := aTempPointers[1]^.stat.lrTempK;
stat.lrSens3TempK := aTempPointers[2]^.stat.lrTempK;
stat.lrSens4TempK := aTempPointers[3]^.stat.lrTempK;
stat.lrSens5TempK := aTempPointers[4]^.stat.lrTempK;

stat.bValidSensor1  := aTempPointers[0]^.stat.bValid;
stat.bValidSensor2  := aTempPointers[1]^.stat.bValid;
stat.bValidSensor3  := aTempPointers[2]^.stat.bValid;
stat.bValidSensor4  := aTempPointers[3]^.stat.bValid;
stat.bValidSensor5  := aTempPointers[4]^.stat.bValid;

// copy some writeable values to the read-only stat struct

stat.sDescription := sDescription;



// If disabled, don't do anything
IF NOT stat.bEnabled THEN
    stat.bValid := FALSE;
    RETURN;
END_IF

//
// If simulated, set the simulated value and return.
// Note: Simulated temperature is in [K] !!!
//

IF in_bSimulation THEN
	stat.bSimulated	:= TRUE;
	stat.bValid		:= TRUE;
	stat.lrTempK	:= stat.lrSimTempK;
	stat.lrTempC	:= stat.lrSimTempK - 273.15;
	RETURN;
ELSE
	stat.bSimulated	:= FALSE;
END_IF


//
// Get the pressure depending on the voting method.
//
CASE stat.nVoteMethod OF
	E_METIS_TEMP_VOTE_METHOD.AVERAGE:
		M_SetStatus_Average();
	E_METIS_TEMP_VOTE_METHOD.LOWEST_TEMPERATURE:
		M_SetStatus_Lowest_Temperature();
	E_METIS_TEMP_VOTE_METHOD.HIGHEST_TEMPERATURE:
		M_SetStatus_Highest_Temperature();
	E_METIS_TEMP_VOTE_METHOD.FIRST_VALID_TEMPERATURE:
		M_SetStatus_FirstValid();
	E_METIS_TEMP_VOTE_METHOD.MEDIAN:
		M_SetStatus_Median();
//	E_METIS_TEMP_VOTE_METHOD.TEMPERATURE_3oo5:
//		M_SetStatus_XooY();
ELSE
	;
END_CASE


//
// If the reading is valid, set the simulated value to it.
// This way, switching from normal to simulation will result in
// no jump in the value.
//
IF stat.bValid  THEN
	stat.lrSimTempK	:= stat.lrTempK;
END_IF

// update also the output data
q_lrTemp := stat.lrTempK;
q_bValid := stat.bValid;
toggleTimer(IN := NOT toggleTimer.Q, PT := T#500ms);
IF toggleTimer.Q AND stat.bValid THEN
    q_bToggle := NOT q_bToggle;
END_IF
END_METHOD

METHOD M_SetStatus_Average
VAR_INPUT
END_VAR
VAR
	lrTmp:		LREAL;	// Temporary var for sum of Temperatures
	nSample:	INT;	// Number of valid sensor readings
	i:			INT;
END_VAR
lrTmp	:= 0.0;
nSample	:= 0;

FOR i:=0 TO 4 DO
	IF aTempIndexes[i] > 0  THEN
		IF aTempPointers[i]^.stat.bValid	THEN
			lrTmp	:= lrTmp + aTempPointers[i]^.stat.lrTempK;
			nSample	:= nSample + 1;
		END_IF
	END_IF
END_FOR

IF nSample > 0	THEN
	stat.lrTempK	:= lrTmp / nSample;
	stat.bValid		:= TRUE;
ELSE
	stat.lrTempK	:= 9999;
	stat.bValid		:= FALSE;
END_IF
END_METHOD

METHOD M_SetStatus_FirstValid
VAR_INPUT
END_VAR
VAR
	lrTmp:		LREAL;	// Temporary var for sum of Temperatures
	nSample:	INT;	// Number of valid sensor readings
	i:			INT;
END_VAR
(*First Valid Temperature*)

nSample	:= 0;

FOR i:=0 TO 4 DO
	IF aTempIndexes[i] > 0  THEN
		IF  aTempPointers[i]^.stat.bValid	THEN
			lrTmp	:= aTempPointers[i]^.stat.lrTempK;
			nSample	:= nSample + 1;
			EXIT;
		END_IF
	END_IF
END_FOR

IF nSample > 0	THEN
	stat.lrTempK	:= lrTmp;
	stat.bValid		:= TRUE;
ELSE
	stat.lrTempK	:= 9999;
	stat.bValid		:= FALSE;
END_IF
END_METHOD

METHOD M_SetStatus_Highest_Temperature
VAR_INPUT
END_VAR
VAR
	lrTmp:		LREAL;	// Temporary var for sum of Temperatures
	nSample:	INT;	// Number of valid sensor readings
	i:			INT;
END_VAR
(*Highest Temperature*)

lrTmp	:= -10000.0; // setting initial temperature for comparision
nSample	:= 0;

FOR i:=0 TO 4 DO
	IF aTempIndexes[i] > 0  THEN
		IF  aTempPointers[i]^.stat.bValid	THEN
				IF  aTempPointers[i]^.stat.lrTempK > lrTmp THEN
					lrTmp	:= aTempPointers[i]^.stat.lrTempK;
				END_IF
			nSample	:= nSample + 1;
		END_IF
	END_IF
END_FOR

IF nSample > 0	THEN
	stat.lrTempK	:= lrTmp;
	stat.bValid		:= TRUE;
ELSE
	stat.lrTempK	:= 9999;
	stat.bValid		:= FALSE;
END_IF
END_METHOD

METHOD M_SetStatus_Lowest_Temperature
VAR_INPUT
END_VAR
VAR
	lrTmp:		LREAL;	// Temporary var for sum of Temperatures
	nSample:	INT;	// Number of valid sensor readings
	i:			INT;
END_VAR
(*Lowest Temperature*)

lrTmp	:= 10000.0; // setting initial temperature for comparision
nSample	:= 0;

FOR i:=0 TO 4 DO
	IF aTempIndexes[i] > 0  THEN
		IF  aTempPointers[i]^.stat.bValid	THEN
				IF  aTempPointers[i]^.stat.lrTempK < lrTmp THEN
					lrTmp	:= aTempPointers[i]^.stat.lrTempK;
				END_IF
			nSample	:= nSample + 1;
		END_IF
	END_IF
END_FOR

IF nSample > 0	THEN
	stat.lrTempK	:= lrTmp;
	stat.bValid		:= TRUE;
ELSE
	stat.lrTempK	:= 9999;
	stat.bValid		:= FALSE;
END_IF
END_METHOD

METHOD M_SetStatus_Median
VAR_INPUT
END_VAR
VAR
    lrTmpArray: ARRAY[0..4] OF LREAL; // Array to store valid temperatures
    nSample:    INT;                // Number of valid sensor readings
    i:          INT;
    j:          INT;
    lrTemp:     LREAL;             // Temporary variable for swapping
END_VAR
nSample := 0;

// Store valid temperatures in the array
FOR i := 0 TO 4 DO
    IF aTempIndexes[i] > 0 THEN
        IF aTempPointers[i]^.stat.bValid THEN
            lrTmpArray[nSample] := aTempPointers[i]^.stat.lrTempK;
            nSample := nSample + 1;
        END_IF
    END_IF
END_FOR

// Sort the array in ascending order (using Bubble Sort for simplicity)
IF nSample > 1 THEN
    FOR i := 0 TO nSample - 2 DO
        FOR j := i + 1 TO nSample - 1 DO
            IF lrTmpArray[i] > lrTmpArray[j] THEN
                lrTemp := lrTmpArray[i];
                lrTmpArray[i] := lrTmpArray[j];
                lrTmpArray[j] := lrTemp;
            END_IF
        END_FOR
    END_FOR
END_IF

// Calculate the median
IF nSample > 0 THEN
    IF nSample MOD 2 = 1 THEN // Odd number of elements
        stat.lrTempK := lrTmpArray[nSample / 2];
    ELSE // Even number of elements
        stat.lrTempK := (lrTmpArray[nSample / 2 - 1] + lrTmpArray[nSample / 2]) / 2.0;
    END_IF
    stat.bValid := TRUE;
ELSE
    stat.lrTempK := 9999;
    stat.bValid := FALSE;
END_IF
END_METHOD

// Calculate pressure based on the status of the two sensors
METHOD M_SetStatus_XooY
//VAR_INPUT
//	in_nNum:	INT;	// Number of readings to select for voting (X)
//	in_nTotal:	INT;	// Total number of readings to check (Y)
//END_VAR
//VAR
//	idx_i, idx_j:	INT;
//	nTmp:		INT;			// Temporary INT var
//	lrTmp:		LREAL	:= 0.0;	// Temporary var for sum of pressures
//	nValid:		INT		:= 0;	// Total number of valid readings
//	nSample:	INT		:= 0;	// Number of valid sensor readings
	
//	aDiff:		ARRAY [1..5,1..5] OF LREAL;	// Table of absolute differences
//	aDiffSum:	ARRAY [1..5] OF LREAL;		// Array of sums of absolute differences
//	// Array of indexes of sums of absolute differences
//	aDiffSumIdx:ARRAY [1..5] OF INT := [1,2,3,4,5];		
//	lrAbsDiff:	LREAL;						// Absolute difference between two readings
	
//	i:			INT;
//	j:			INT;
//END_VAR
VAR
	lrTmp:		LREAL;	// Temporary var for sum of Temperatures
	nSample:	INT;	// Number of valid sensor readings
	i:			INT;
END_VAR
(*Average Temperature*)

lrTmp	:= 0.0;
nSample	:= 0;

FOR i:=0 TO 4 DO
	IF aTempIndexes[i] > 0  THEN
		IF  aTempPointers[i]^.stat.bValid	THEN
			lrTmp	:= lrTmp + aTempPointers[i]^.stat.lrTempK;
			nSample	:= nSample + 1;
		END_IF
	END_IF
END_FOR

IF nSample > 0	THEN
	stat.lrTempK	:= lrTmp / nSample;
	stat.bValid		:= TRUE;
ELSE
	stat.lrTempK	:= 9999;
	stat.bValid		:= FALSE;
END_IF








////
////	Get the number of valid readings and calculate the average
////
//FOR i:=1 TO in_nTotal DO
//	IF pSensor[i] <> 0  THEN
//		IF  pSensor[i]^.stat.bValid	THEN
//			lrTmp	:= lrTmp + pSensor[i]^.stat.lrPressure;
//			nValid	:= nValid + 1;
//		END_IF
//	END_IF
//END_FOR


////
//// Vote X out of Y
////
//IF nValid >= in_nNum	THEN
//	//
//	// Calculate relative differences between two readings, 
//	// relative to the bigger ABS value.
//	// Table is symetric. Calculate only the half (triangle) on the right. 
//	// Make a copy to the other half.
//	//
//	FOR i:=1 TO in_nTotal DO
//		FOR j:=i+1 TO in_nTotal DO
//			IF pSensor[i] <> 0  AND  pSensor[j] <> 0	THEN
//				IF pSensor[i]^.stat.bValid  AND  pSensor[j]^.stat.bValid	THEN
//					lrAbsDiff	:= ABS(pSensor[i]^.stat.lrPressure - pSensor[j]^.stat.lrPressure);
//					aDiff[i,j]	:= lrAbsDiff;
//					aDiff[j,i]	:= lrAbsDiff;
//				ELSE
//					aDiff[i,j]	:= 9999.0;
//					aDiff[j,i]	:= 9999.0;
//				END_IF
//			ELSE
//				aDiff[i,j]	:= 9999.0;
//				aDiff[j,i]	:= 9999.0;
//			END_IF
//		END_FOR
//	END_FOR

//	//
//	// Get the sum of all differences for each reading.
//	//
//	FOR i:=1 TO in_nTotal DO
//		aDiffSum[i]	:= 0.0;
//		FOR j:=1 TO in_nTotal DO
//			aDiffSum[i]	:= aDiffSum[i] + aDiff[i,j];
//		END_FOR
//	END_FOR

//	//
//	// Sort the indexes for differences in accending order (low sum first).
//	//
//	FOR i:=1 TO in_nTotal DO
//		FOR j:=i+1 TO in_nTotal DO
//			idx_i	:= aDiffSumIdx[i];
//			idx_j	:= aDiffSumIdx[j];
//			IF aDiffSum[idx_j] < aDiffSum[idx_i]	THEN
//				// Swap indexes
//				nTmp			:= aDiffSumIdx[j];
//				aDiffSumIdx[j]	:= aDiffSumIdx[i];
//				aDiffSumIdx[i]	:= nTmp;
//			END_IF
//		END_FOR
//	END_FOR

	
//	//					
//	// Get the average of selected in_nNum readings.
//	// Assign the result to the pressure.
//	//
//	lrTmp	:= 0.0;
//	FOR i:=1 TO in_nNum DO
//		idx_i	:= aDiffSumIdx[i];
//		lrTmp	:= lrTmp + pSensor[idx_i]^.stat.lrPressure;
//	END_FOR
	
//	stat.lrPressure	:= lrTmp / in_nNum;
//	stat.bValid		:= TRUE;
//ELSE
//	stat.lrPressure	:= 9999;
//	stat.bValid		:= FALSE;
//END_IF
END_METHOD

METHOD M_UpdateTempPointers
VAR_INPUT
END_VAR
VAR_IN_OUT
    met_temp : FB_METIS_TEMPERATURES;
END_VAR
VAR 
    i : INT;
END_VAR
FOR i := 0 TO 4 DO
    aTempPointers[i] := met_temp.M_SetTemperatureSensor(TO_INT(aTempIndexes[i]));
END_FOR


IF NOT bConfigured THEN
    M_Configure(met_temp := met_temp);
    RETURN;
END_IF
END_METHOD

END_FUNCTION_BLOCK

// POUs/Routines/CabinetControl/FB_METIS_CABINET_CTRL
FUNCTION_BLOCK FB_METIS_CABINET_CTRL
VAR_INPUT
END_VAR
VAR_OUTPUT
END_VAR
VAR
END_VAR

END_FUNCTION_BLOCK

// HMI/VISUs/Cryo_Devices/Cabinets/VISU_HMI_CABINETS
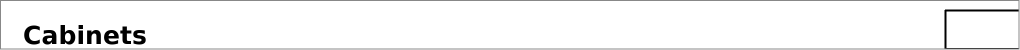
VISUALIZATION VISU_HMI_CABINETS  // 1020x50
    Label (20,20 163x30), "Cabinets"
    Frame (945,10 75x40)
        shows VISU_HMI_SUBSYSTEM_BUTTON(m_Hmi := PRG_HMI.fbBackButton)
        OnMouseClick: execute { PRG_HMI.eActiveTab := PRG_HMI.ePreviousTab; }
END_VISUALIZATION

// HMI/VISUs/Cryo_Devices/Control_Loops/VISU_HMI_CONTROL_LOOPS
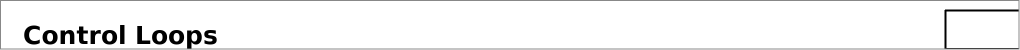
VISUALIZATION VISU_HMI_CONTROL_LOOPS  // 1020x50
    Label (20,20 208x30), "Control Loops"
    Frame (945,10 75x40)
        shows VISU_HMI_SUBSYSTEM_BUTTON(m_Hmi := PRG_HMI.fbBackButton)
        OnMouseClick: execute { PRG_HMI.eActiveTab := PRG_HMI.ePreviousTab; }
END_VISUALIZATION

// HMI/VISUs/Cryo_Devices/Control_Units/VISU_HMI_CONTROL_UNITS
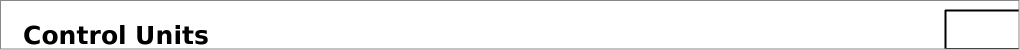
VISUALIZATION VISU_HMI_CONTROL_UNITS  // 1020x50
    Label (20,20 187x30), "Control Units"
    Frame (945,10 75x40)
        shows VISU_HMI_SUBSYSTEM_BUTTON(m_Hmi := PRG_HMI.fbBackButton)
        OnMouseClick: execute { PRG_HMI.eActiveTab := PRG_HMI.ePreviousTab; }
END_VISUALIZATION

// HMI/VISUs/Cryo_Devices/Coolers/VISU_HMI_COOLERS
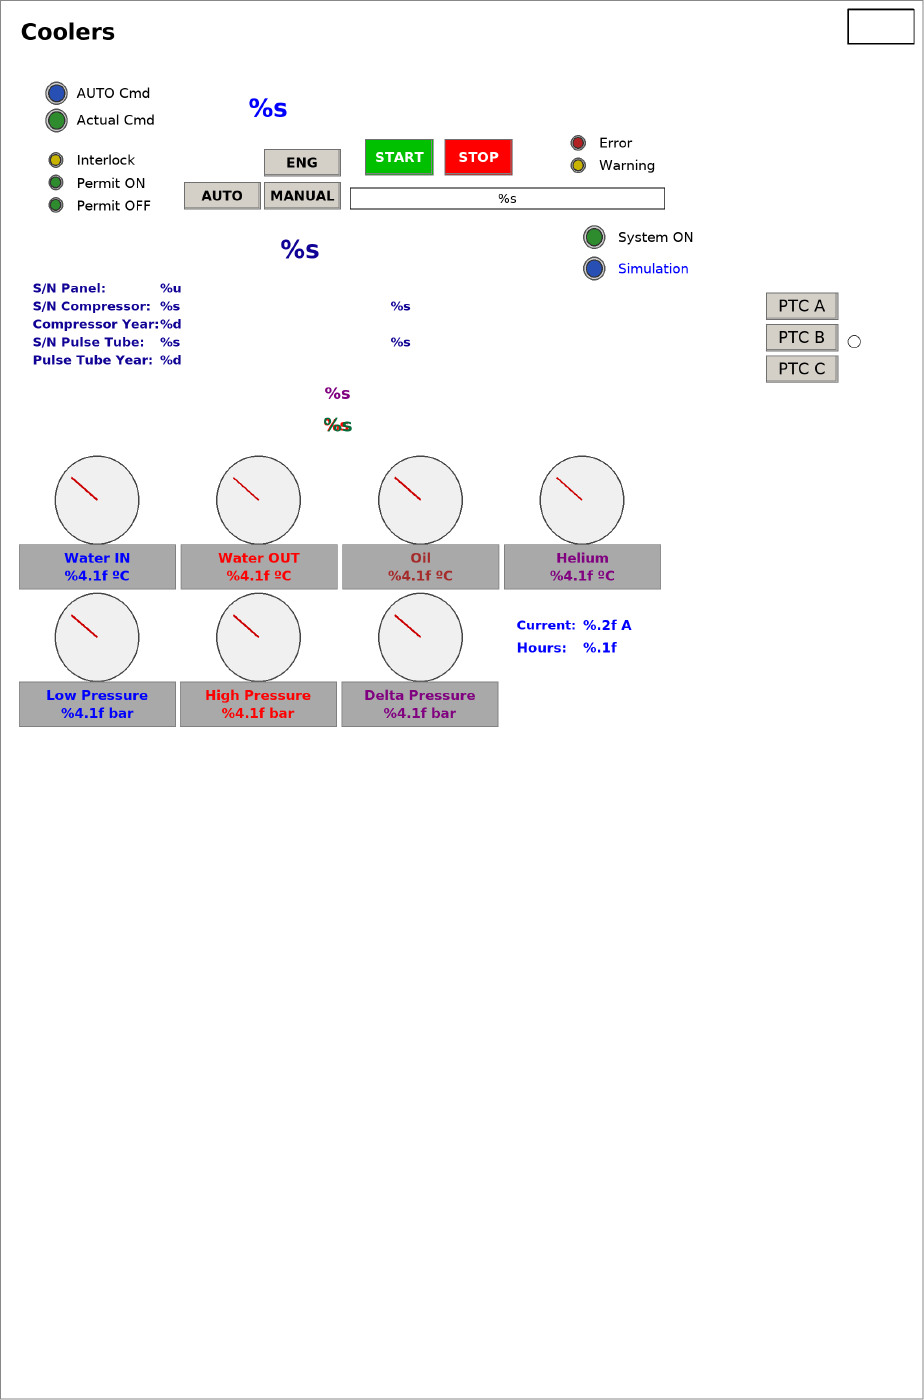
VISUALIZATION VISU_HMI_COOLERS  // 1030x1560
    Label (20,20 163x30), "Coolers"
    Frame (10,63 773x747)
        shows TEMPLATE_METIS_CRYO_CPA(m_Instance := MAIN.met_cryo_ctrl.met_cool_down.ptc[MAIN.met_cryo_ctrl.met_cool_down.guiIndex_cor_ptcs], m_Cmd := MAIN.met_cryo_ctrl.met_cool_down.ptrArr_cor_ptcs[MAIN.met_cryo_ctrl.met_cool_down.guiIndex_cor_ptcs]^)
    Button (854,326 80x30), "PTC A", tooltip "Pulse Tube Cooler A"
        OnMouseClick: execute { MAIN.met_cryo_ctrl.met_cool_down.guiIndex_cor_ptcs := 1; }
    Button (854,361 80x30), "PTC B", tooltip "Pulse Tube Cooler B"
        OnMouseClick: execute { MAIN.met_cryo_ctrl.met_cool_down.guiIndex_cor_ptcs := 2; }
    Button (854,396 80x30), "PTC C", tooltip "Pulse Tube Cooler C"
        OnMouseClick: execute { MAIN.met_cryo_ctrl.met_cool_down.guiIndex_cor_ptcs := 3; }
    RadioButton (943,329 57x103), variable: MAIN.met_cryo_ctrl.met_cool_down.guiIndex_cor_ptcs-1
        Areas[0]: Text=Radiobutton
        Areas[1]: Text=Radiobutton
    Frame (945,10 75x40)
        shows VISU_HMI_SUBSYSTEM_BUTTON(m_Hmi := PRG_HMI.fbBackButton)
        OnMouseClick: execute { PRG_HMI.eActiveTab := PRG_HMI.ePreviousTab; }
END_VISUALIZATION

// HMI/VISUs/Cryo_Devices/Detectors/VISU_HMI_DETECTORS
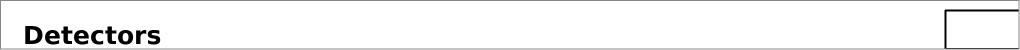
VISUALIZATION VISU_HMI_DETECTORS  // 1020x50
    Label (20,20 163x30), "Detectors"
    Frame (945,10 75x40)
        shows VISU_HMI_SUBSYSTEM_BUTTON(m_Hmi := PRG_HMI.fbBackButton)
        OnMouseClick: execute { PRG_HMI.eActiveTab := PRG_HMI.ePreviousTab; }
END_VISUALIZATION

// HMI/VISUs/Cryo_Devices/Heaters/VISU_HMI_HEATERS
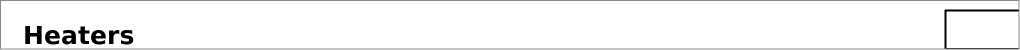
VISUALIZATION VISU_HMI_HEATERS  // 1020x50
    Label (20,20 163x30), "Heaters"
    Frame (945,10 75x40)
        shows VISU_HMI_SUBSYSTEM_BUTTON(m_Hmi := PRG_HMI.fbBackButton)
        OnMouseClick: execute { PRG_HMI.eActiveTab := PRG_HMI.ePreviousTab; }
END_VISUALIZATION

// HMI/VISUs/Cryo_Devices/Pressures/VISU_HMI_PRESSURES
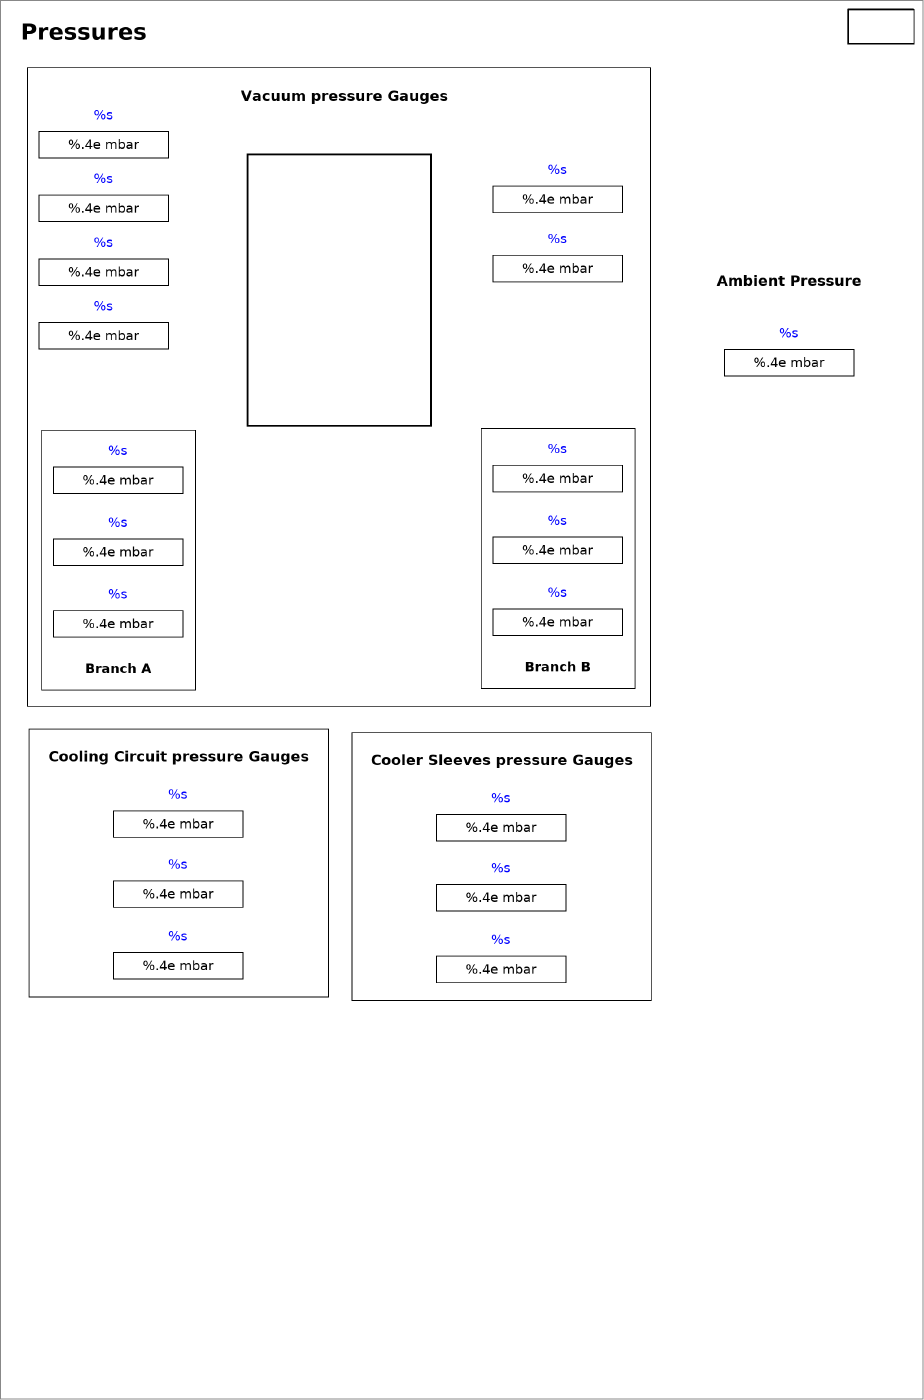
VISUALIZATION VISU_HMI_PRESSURES  // 1030x1560
    Rectangle (30,75 695x712)
    Rectangle (32,812 334x299)
    Label (20,20 163x30), "Pressures"
    Group (41,111 150x283)
        Frame (0,0 150x70)
            shows TEMPLATE_PRESSURE_READING(m_instance := MAIN.met_cryo_ctrl.met_evac.sensor_VAGF1)
        Frame (0,71 150x70)
            shows TEMPLATE_PRESSURE_READING(m_instance := MAIN.met_cryo_ctrl.met_evac.sensor_VAGF2)
        Frame (0,142 150x70)
            shows TEMPLATE_PRESSURE_READING(m_instance := MAIN.met_cryo_ctrl.met_evac.sensor_VAGG1)
        Frame (0,213 150x70)
            shows TEMPLATE_PRESSURE_READING(m_instance := MAIN.met_cryo_ctrl.met_evac.sensor_VAGG2)
    Group (547,172 150x147)
        Frame (0,0 150x70)
            shows TEMPLATE_PRESSURE_READING(m_instance := MAIN.met_cryo_ctrl.met_venting.sensor_HPG1)
        Frame (0,77 150x70)
            shows TEMPLATE_PRESSURE_READING(m_instance := MAIN.met_cryo_ctrl.met_venting.sensor_HPG2)
    Frame (124,868 150x70)
        shows TEMPLATE_PRESSURE_READING(m_instance := MAIN.met_cryo_ctrl.met_cool_down.sensor_VAG_P1)
    Frame (124,946 150x70)
        shows TEMPLATE_PRESSURE_READING(m_instance := MAIN.met_cryo_ctrl.met_cool_down.sensor_VAG_PCA)
    Frame (124,1026 150x70)
        shows TEMPLATE_PRESSURE_READING(m_instance := MAIN.met_cryo_ctrl.met_cool_down.sensor_VAG_PCB)
    Group (46,479 172x290)
        Rectangle (0,0 172x290)
        Group (11,6 150x275)
            Frame (0,0 150x70)
                shows TEMPLATE_PRESSURE_READING(m_instance := MAIN.met_cryo_ctrl.met_evac.evac_branch_a.sensor_VAG1)
            Frame (0,80 150x70)
                shows TEMPLATE_PRESSURE_READING(m_instance := MAIN.met_cryo_ctrl.met_evac.evac_branch_a.sensor_VAG2)
            Frame (0,160 150x70)
                shows TEMPLATE_PRESSURE_READING(m_instance := MAIN.met_cryo_ctrl.met_evac.evac_branch_a.sensor_VAG3)
            Rectangle (0,245 150x30), "Branch A"
    Group (536,477 172x290)
        Rectangle (0,0 172x290)
        Group (11,6 150x275)
            Frame (0,0 150x70)
                shows TEMPLATE_PRESSURE_READING(m_instance := MAIN.met_cryo_ctrl.met_evac.evac_branch_b.sensor_VAG1)
            Frame (0,80 150x70)
                shows TEMPLATE_PRESSURE_READING(m_instance := MAIN.met_cryo_ctrl.met_evac.evac_branch_b.sensor_VAG2)
            Frame (0,160 150x70)
                shows TEMPLATE_PRESSURE_READING(m_instance := MAIN.met_cryo_ctrl.met_evac.evac_branch_b.sensor_VAG3)
            Rectangle (0,245 150x30), "Branch B"
    Group (260,92 248x383)
        RoundedRectangle (15,79 206x304)
        Rectangle (0,0 248x30), "Vacuum pressure Gauges"
    Rectangle (47,828 305x30), "Cooling Circuit pressure Gauges"
    Rectangle (392,816 334x299)
    Frame (484,872 150x70)
        shows TEMPLATE_PRESSURE_READING(m_instance := MAIN.met_cryo_ctrl.sensor_VAG_PTA)
    Frame (484,950 150x70)
        shows TEMPLATE_PRESSURE_READING(m_instance := MAIN.met_cryo_ctrl.sensor_VAG_PTB)
    Frame (484,1030 150x70)
        shows TEMPLATE_PRESSURE_READING(m_instance := MAIN.met_cryo_ctrl.sensor_VAG_PTC)
    Rectangle (407,832 305x30), "Cooler Sleeves pressure Gauges"
    Frame (945,10 75x40)
        shows VISU_HMI_SUBSYSTEM_BUTTON(m_Hmi := PRG_HMI.fbBackButton)
        OnMouseClick: execute { PRG_HMI.eActiveTab := PRG_HMI.ePreviousTab; }
    Frame (805,354 150x70)
        shows TEMPLATE_AMBIENT_PRESSURE_READING(m_instance := MAIN.met_cryo_ctrl.sensor_AMB_PRESS)
    Rectangle (765,298 230x30), "Ambient Pressure"
END_VISUALIZATION

// HMI/VISUs/Cryo_Devices/Pumps/VISU_HMI_PUMPS
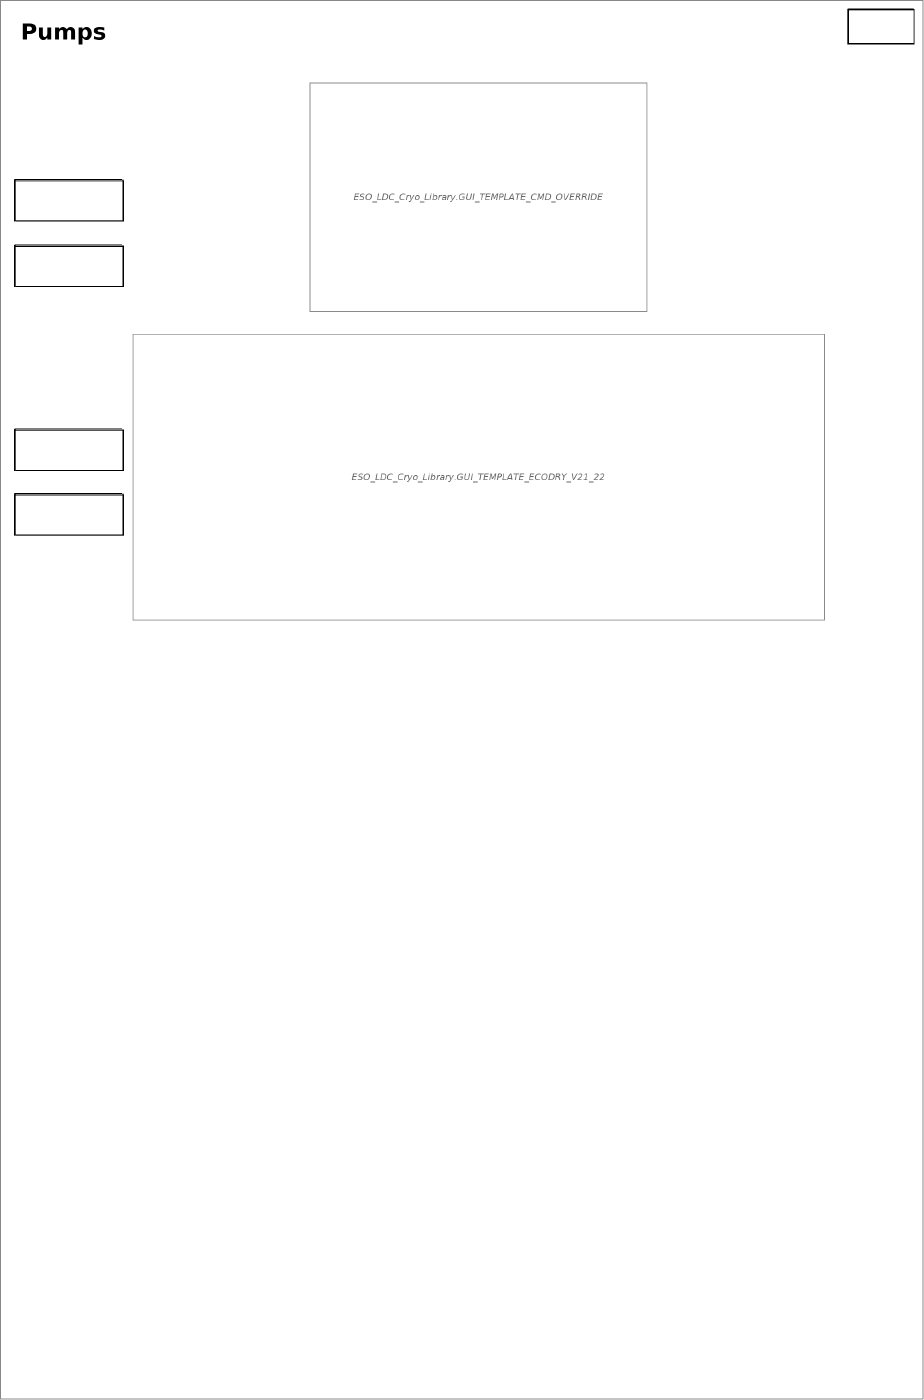
VISUALIZATION VISU_HMI_PUMPS  // 1030x1560
VAR_IN_OUT
	m_Hmi:		FB_HMI_PUMPS;
END_VAR
    Label (20,20 163x30), "Pumps"
    Frame (148,92 850x800), frame switch variable: m_Hmi.eActiveTab
        shows VISU_HMI_RP_BRANCH_A()
        shows VISU_HMI_TP_BRANCH_A()
        shows VISU_HMI_RP_BRANCH_B()
        shows VISU_HMI_TP_BRANCH_B()
    Frame (16,200 123x48)
        shows VISU_HMI_SUBSYSTEM_BUTTON(m_Hmi := m_Hmi.fbRpBranchAButton)
        OnMouseClick: execute { m_Hmi.eActiveTab := E_HMI_PUMPS_TABS.RP_BRANCH_A; }
    Frame (16,273 123x48)
        shows VISU_HMI_SUBSYSTEM_BUTTON(m_Hmi := m_Hmi.fbTpBranchAButton)
        OnMouseClick: execute { m_Hmi.eActiveTab := E_HMI_PUMPS_TABS.TP_BRANCH_A; }
    Frame (16,478 123x48)
        shows VISU_HMI_SUBSYSTEM_BUTTON(m_Hmi := m_Hmi.fbRpBranchBButton)
        OnMouseClick: execute { m_Hmi.eActiveTab := E_HMI_PUMPS_TABS.RP_BRANCH_B; }
    Frame (16,550 123x48)
        shows VISU_HMI_SUBSYSTEM_BUTTON(m_Hmi := m_Hmi.fbTpBranchBButton)
        OnMouseClick: execute { m_Hmi.eActiveTab := E_HMI_PUMPS_TABS.TP_BRANCH_B; }
    Frame (945,10 75x40)
        shows VISU_HMI_SUBSYSTEM_BUTTON(m_Hmi := PRG_HMI.fbBackButton)
        OnMouseClick: execute { PRG_HMI.eActiveTab := PRG_HMI.ePreviousTab; }
END_VISUALIZATION

// HMI/VISUs/Cryo_Devices/Pumps/VISU_HMI_RP_BRANCH_A
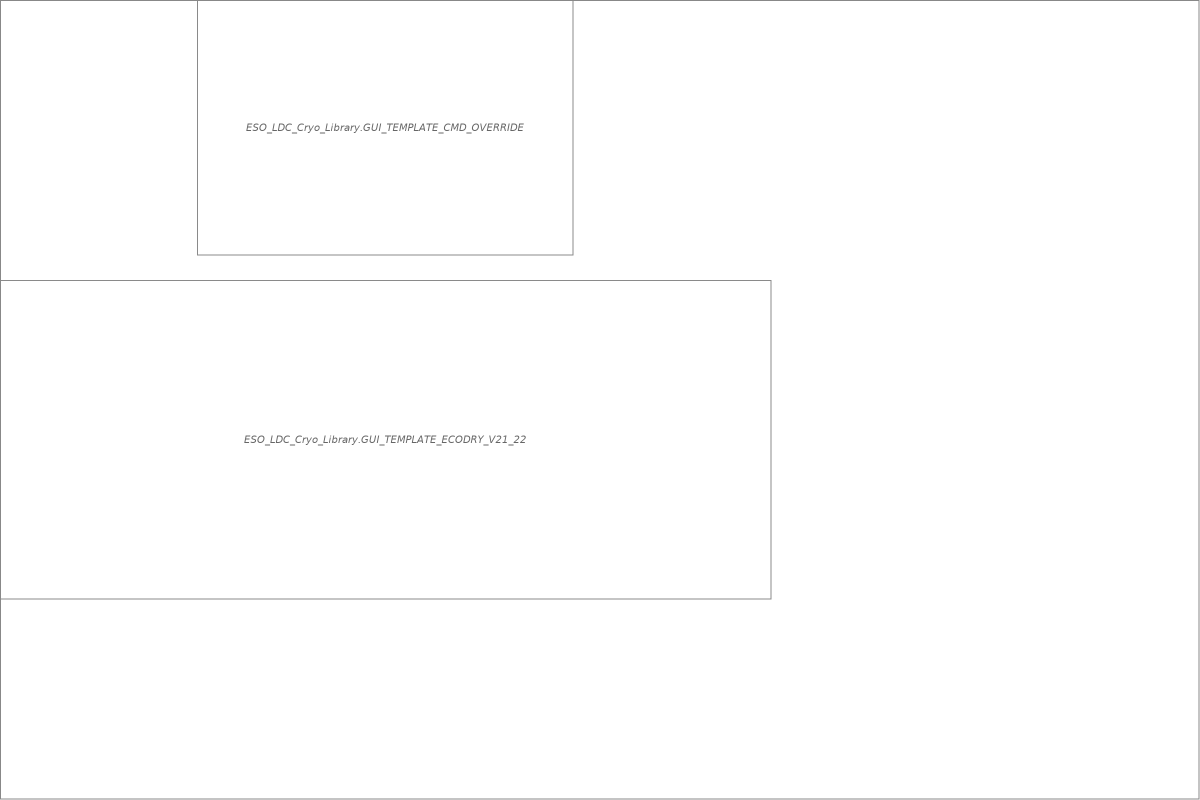
VISUALIZATION VISU_HMI_RP_BRANCH_A  // 1200x800
    Group (0,0 771x599)
        Frame (0,280 771x319)
            shows ESO_LDC_Cryo_Library.GUI_TEMPLATE_ECODRY_V21_22(m_Instance := MAIN.met_cryo_ctrl.met_evac.evac_branch_a.rp, m_bEnable := MAIN.met_cryo_ctrl.met_evac.evac_branch_a.rp.in_bEnable)
        Frame (197,0 376x255)
            shows ESO_LDC_Cryo_Library.GUI_TEMPLATE_CMD_OVERRIDE(m_Cmd := MAIN.met_cryo_ctrl.met_evac.evac_branch_a.cor_rp)
END_VISUALIZATION

// HMI/VISUs/Cryo_Devices/Pumps/VISU_HMI_RP_BRANCH_B
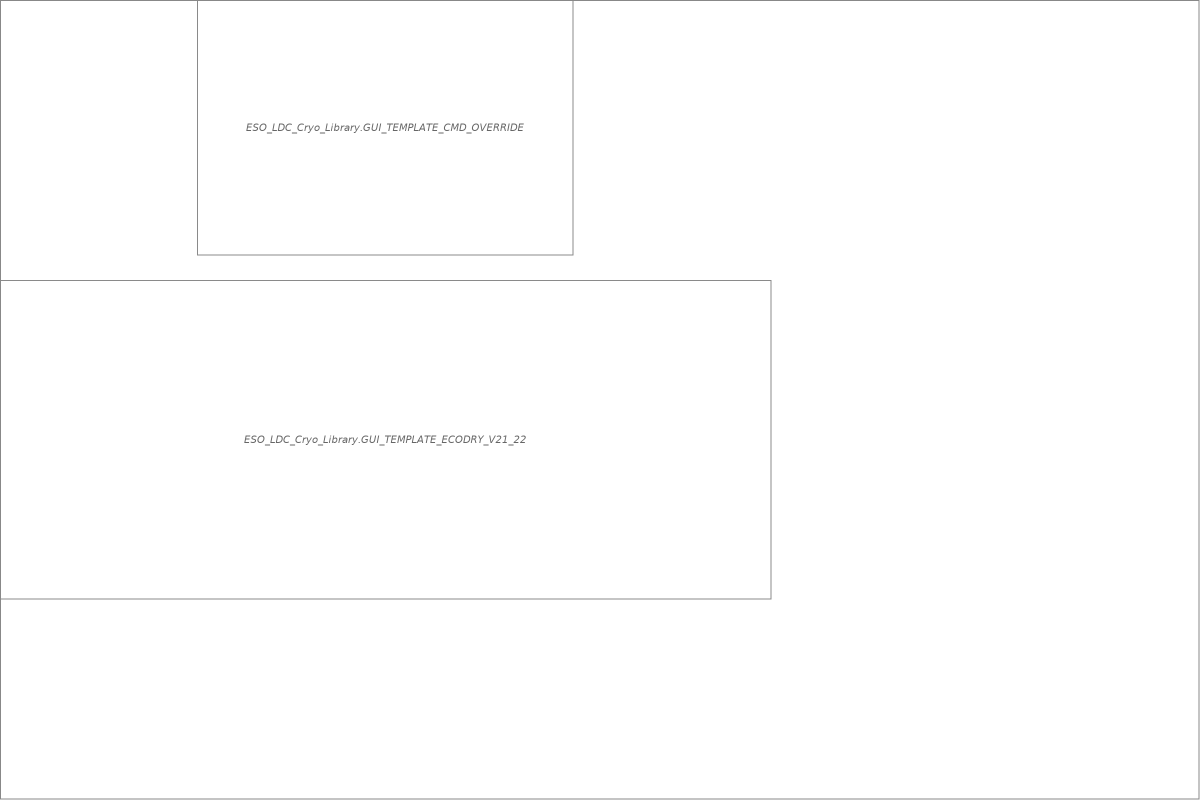
VISUALIZATION VISU_HMI_RP_BRANCH_B  // 1200x800
    Group (0,0 771x599)
        Frame (0,280 771x319)
            shows ESO_LDC_Cryo_Library.GUI_TEMPLATE_ECODRY_V21_22(m_Instance := MAIN.met_cryo_ctrl.met_evac.evac_branch_b.rp, m_bEnable := MAIN.met_cryo_ctrl.met_evac.evac_branch_b.rp.in_bEnable)
        Frame (197,0 376x255)
            shows ESO_LDC_Cryo_Library.GUI_TEMPLATE_CMD_OVERRIDE(m_Cmd := MAIN.met_cryo_ctrl.met_evac.evac_branch_b.cor_rp)
END_VISUALIZATION

// HMI/VISUs/Cryo_Devices/Pumps/VISU_HMI_TP_BRANCH_A
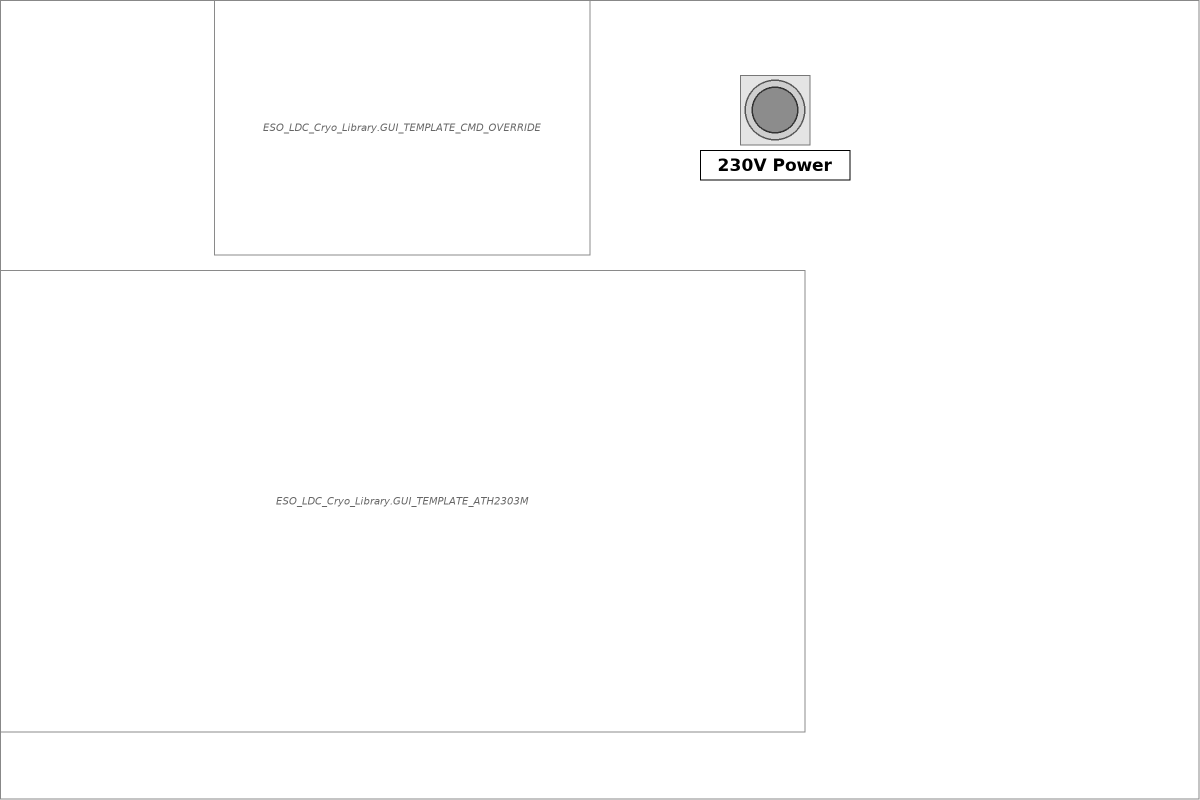
VISUALIZATION VISU_HMI_TP_BRANCH_A  // 1200x800
    Group (0,0 805x732)
        Frame (0,270 805x462)
            shows ESO_LDC_Cryo_Library.GUI_TEMPLATE_ATH2303M(m_Instance := MAIN.met_cryo_ctrl.met_evac.evac_branch_a.tp, m_bEnable := MAIN.met_cryo_ctrl.met_evac.evac_branch_a.tp.in_bEnable)
        Frame (214,0 376x255)
            shows ESO_LDC_Cryo_Library.GUI_TEMPLATE_CMD_OVERRIDE(m_Cmd := MAIN.met_cryo_ctrl.met_evac.evac_branch_a.cor_tp)
    Group (700,75 150x105)
        Rectangle (0,75 150x30), "230V Power", tooltip "Mains power supply"
        PushSwitchLed (40,0 70x70), variable: MAIN.met_cryo_ctrl.met_evac.bTP_A_pwr, behaviour: TOGGLE, style: Switch-PushSwitchLed-Gray
END_VISUALIZATION

// HMI/VISUs/Cryo_Devices/Pumps/VISU_HMI_TP_BRANCH_B
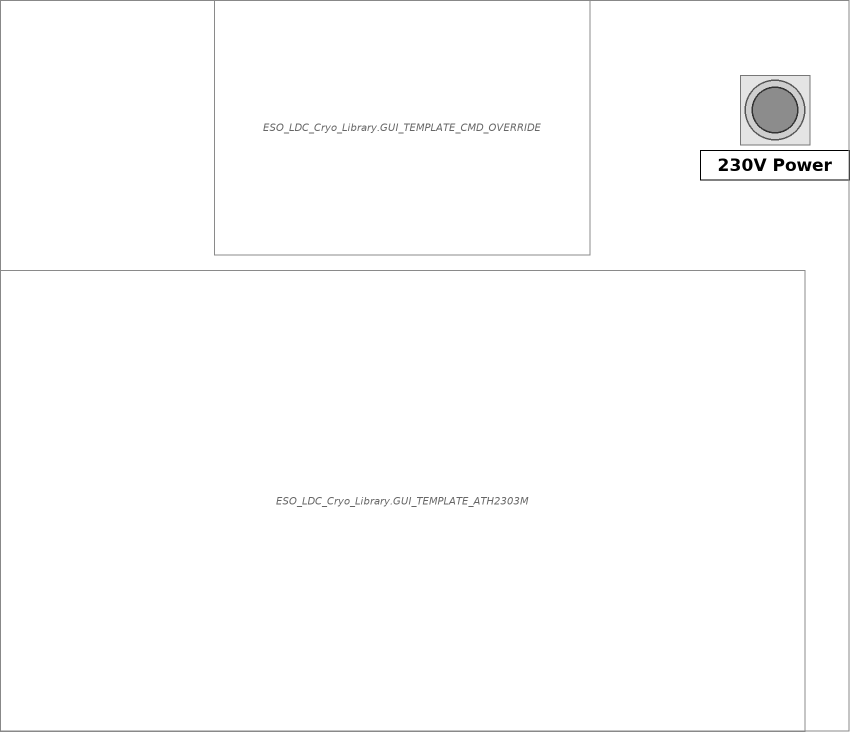
VISUALIZATION VISU_HMI_TP_BRANCH_B  // 850x732
    Group (0,0 805x732)
        Frame (0,270 805x462)
            shows ESO_LDC_Cryo_Library.GUI_TEMPLATE_ATH2303M(m_Instance := MAIN.met_cryo_ctrl.met_evac.evac_branch_b.tp, m_bEnable := MAIN.met_cryo_ctrl.met_evac.evac_branch_b.tp.in_bEnable)
        Frame (214,0 376x255)
            shows ESO_LDC_Cryo_Library.GUI_TEMPLATE_CMD_OVERRIDE(m_Cmd := MAIN.met_cryo_ctrl.met_evac.evac_branch_b.cor_tp)
    Group (700,75 150x105)
        Rectangle (0,75 150x30), "230V Power", tooltip "Mains power supply"
        PushSwitchLed (40,0 70x70), variable: MAIN.met_cryo_ctrl.met_evac.bTP_B_pwr, behaviour: TOGGLE, style: Switch-PushSwitchLed-Gray
END_VISUALIZATION

// HMI/VISUs/Cryo_Devices/Temperatures/Components/VISU_HMI_SYSTEM_VOTERS
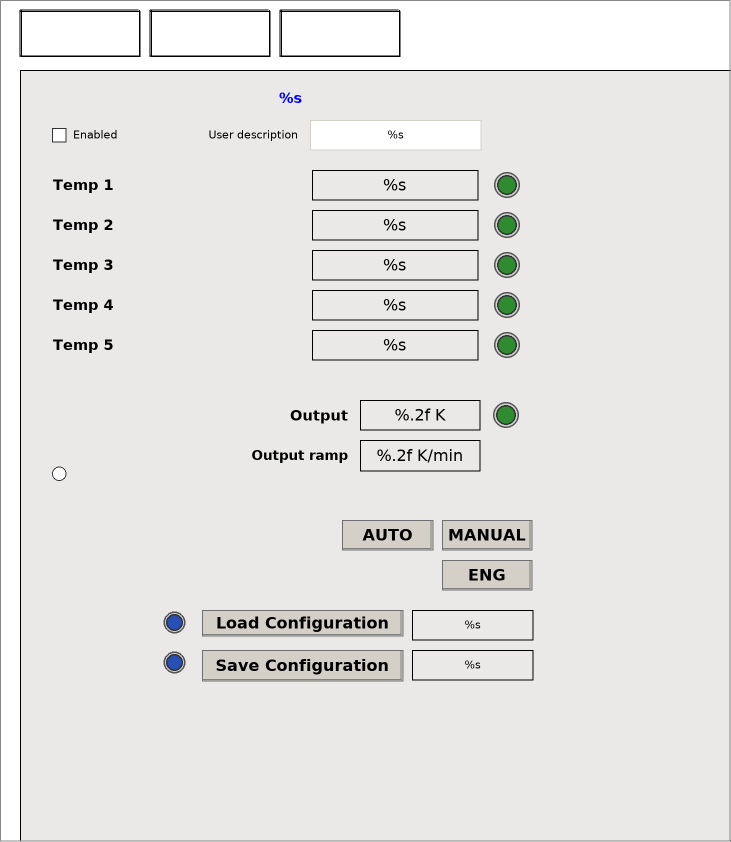
VISUALIZATION VISU_HMI_SYSTEM_VOTERS  // 731x842
VAR_IN_OUT
    m_Instance : FB_METIS_VOTERS;
	m_Hmi : FB_HMI_TEMP_VOTERS;
    m_temperatures : FB_METIS_TEMPERATURES;
END_VAR
    Frame (0,0 717x842), frame switch variable: m_Hmi.eActiveTab
        shows TEMPLATE_BACKGROUND_LEVEL_3()
    Frame (20,10 121x48)
        shows VISU_HMI_SUBSYSTEM_BUTTON(m_Hmi := m_Hmi.fbVoter1Button)
        OnMouseClick: execute { m_Hmi.eActiveTab := E_HMI_VOTER_TABS.VOTER_1; }
    Frame (150,10 121x48)
        shows VISU_HMI_SUBSYSTEM_BUTTON(m_Hmi := m_Hmi.fbVoter2Button)
        OnMouseClick: execute { m_Hmi.eActiveTab := E_HMI_VOTER_TABS.VOTER_2; }
    Frame (280,10 121x48)
        shows VISU_HMI_SUBSYSTEM_BUTTON(m_Hmi := m_Hmi.fbVoter3Button)
        OnMouseClick: execute { m_Hmi.eActiveTab := E_HMI_VOTER_TABS.VOTER_3; }
    Frame (40,80 691x721), frame switch variable: m_Hmi.eActiveTab
        shows TEMPLATE_TEMPERATURE_VOTE(m_Instance := m_Instance.vote_master_temp, m_all_temperatures_array := m_temperatures)
        shows TEMPLATE_TEMPERATURE_VOTE(m_Instance := m_Instance.vote_master_1, m_all_temperatures_array := m_temperatures)
        shows TEMPLATE_TEMPERATURE_VOTE(m_Instance := m_Instance.vote_master_2, m_all_temperatures_array := m_temperatures)
        shows TEMPLATE_TEMPERATURE_VOTE(m_Instance := m_Instance.vote_cry_4, m_all_temperatures_array := m_temperatures)
        shows TEMPLATE_TEMPERATURE_VOTE(m_Instance := m_Instance.vote_cry_5, m_all_temperatures_array := m_temperatures)
        shows TEMPLATE_TEMPERATURE_VOTE(m_Instance := m_Instance.vote_cry_6, m_all_temperatures_array := m_temperatures)
        shows TEMPLATE_TEMPERATURE_VOTE(m_Instance := m_Instance.vote_cry_7, m_all_temperatures_array := m_temperatures)
        shows TEMPLATE_TEMPERATURE_VOTE(m_Instance := m_Instance.vote_cry_8, m_all_temperatures_array := m_temperatures)
        shows TEMPLATE_TEMPERATURE_VOTE(m_Instance := m_Instance.vote_cry_9, m_all_temperatures_array := m_temperatures)
        shows TEMPLATE_TEMPERATURE_VOTE(m_Instance := m_Instance.vote_cry_10, m_all_temperatures_array := m_temperatures)
END_VISUALIZATION

// HMI/VISUs/Cryo_Devices/Temperatures/VISU_HMI_TEMPERATURES
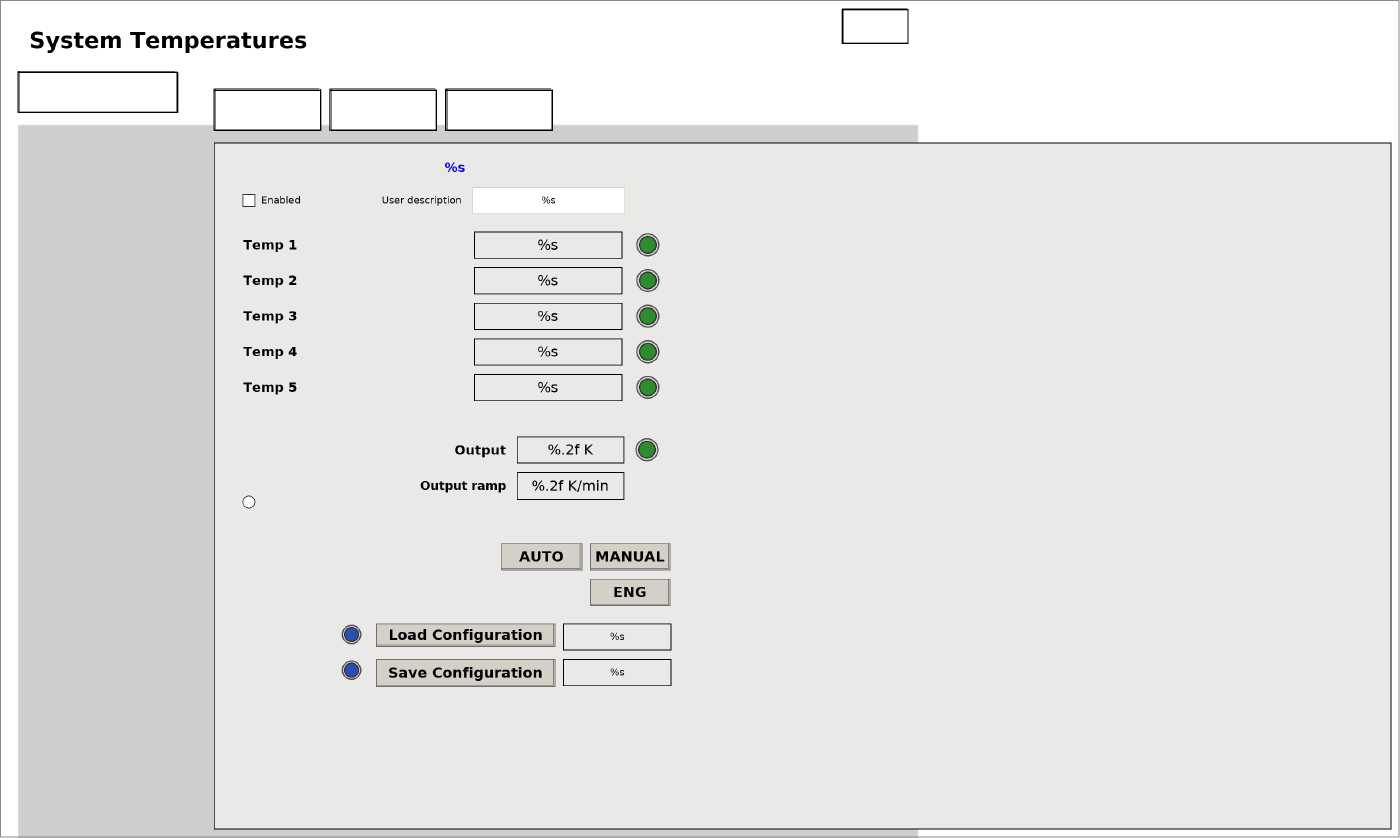
VISUALIZATION VISU_HMI_TEMPERATURES  // 1571x941
VAR_IN_OUT
		met_cryo_ctrl: FB_METIS_CRYO_CTRL;
    	m_Hmi : FB_HMI_TEMPERATURES;
END_VAR
    Frame (10,10 1561x931)
        shows TEMPLATE_BACKGROUND_LEVEL_2()
    Label (30,30 671x30), "System Temperatures"
    Frame (220,90 1191x841), frame switch variable: m_Hmi.eActiveTab
        shows VISU_HMI_SYSTEM_VOTERS(m_Instance := met_cryo_ctrl.met_voters, m_Hmi := m_Hmi.fbVoters, m_temperatures := met_cryo_ctrl.met_temp)
        shows VISU_HMI_CRY_HEATERS(m_Instance := met_cryo_ctrl.met_heaters, m_Hmi := m_Hmi.fbHeaters)
        shows VISU_HMI_CRY_RH(m_Instance := met_cryo_ctrl.met_rh)
        shows VISU_HMI_CRY_VOTERS(m_Instance := met_cryo_ctrl.met_voters, m_Hmi := m_Hmi.fbVoters, m_temperatures := met_cryo_ctrl.met_temp)
        shows VISU_HMI_CRY_TCTRL(m_Instance := met_cryo_ctrl.met_tctrl, m_Hmi := m_Hmi.fbTControl, m_temp := met_cryo_ctrl.met_temp)
        shows VISU_HMI_CRY_LN2_LEVEL_CONTROL()
    Frame (20,80 181x48)
        shows VISU_HMI_SUBSYSTEM_BUTTON(m_Hmi := m_Hmi.fbVotersButton)
        OnMouseClick: execute { m_Hmi.eActiveTab := E_HMI_TEMP_TABS.VOTERS; }
    Frame (945,10 75x40)
        shows VISU_HMI_SUBSYSTEM_BUTTON(m_Hmi := PRG_HMI.fbBackButton)
        OnMouseClick: execute { PRG_HMI.eActiveTab := PRG_HMI.ePreviousTab; }
END_VISUALIZATION

// HMI/VISUs/Cryo_Devices/Valves/VISU_HMI_VALVES
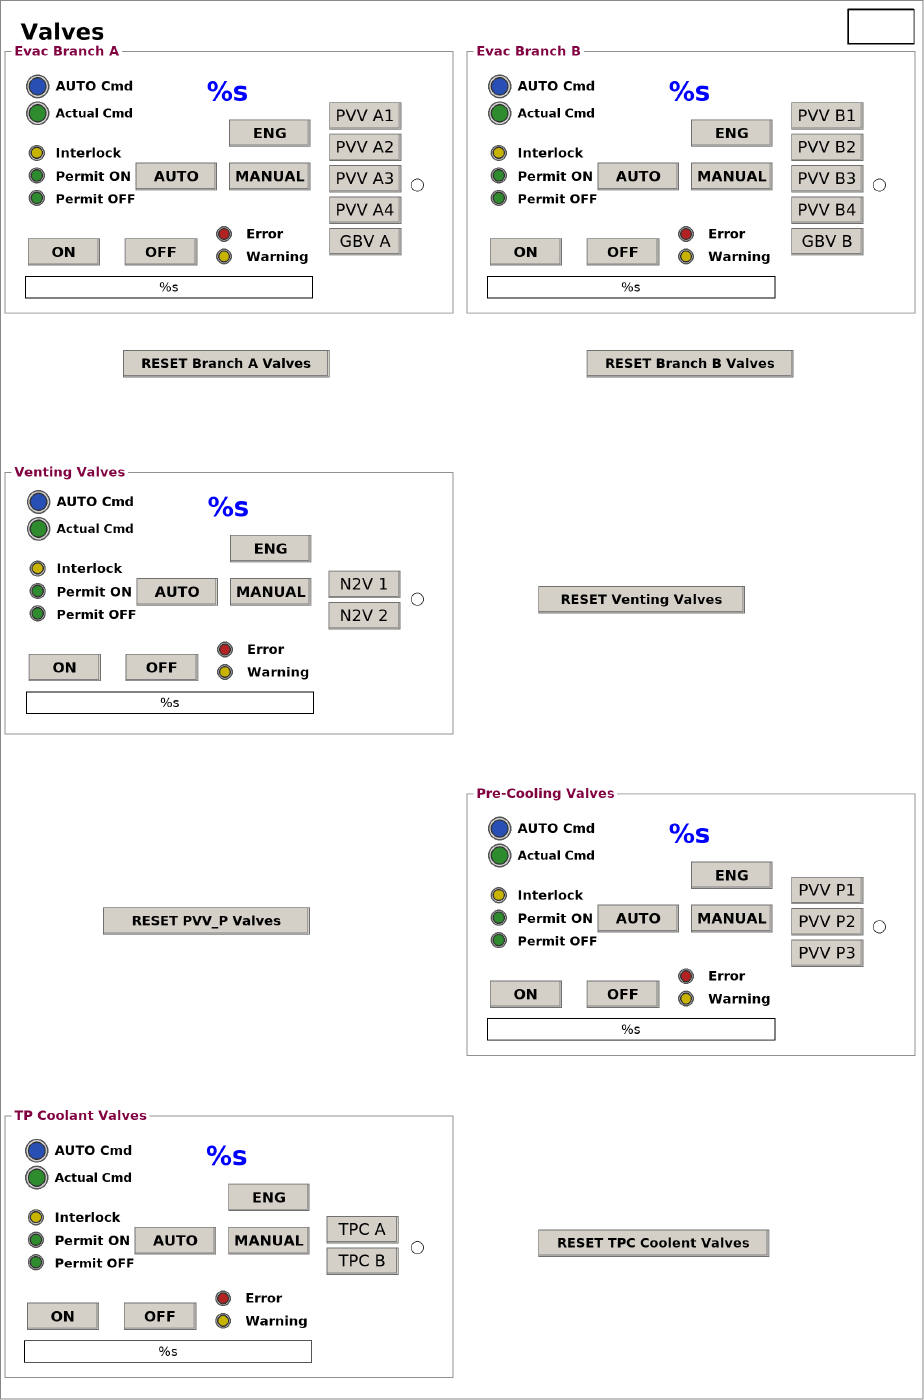
VISUALIZATION VISU_HMI_VALVES  // 1030x1560
    Label (20,20 163x30), "Valves"
    Frame (0,44 1013x1493)
        shows TEMPLATE_BINARY_VALVES(m_evac_Instance := MAIN.met_cryo_ctrl.met_evac, m_venting_instance := MAIN.met_cryo_ctrl.met_venting, m_cool_down_instance := MAIN.met_cryo_ctrl.met_cool_down, m_cryo_instance := MAIN.met_cryo_ctrl)
    Frame (945,10 75x40)
        shows VISU_HMI_SUBSYSTEM_BUTTON(m_Hmi := PRG_HMI.fbBackButton)
        OnMouseClick: execute { PRG_HMI.eActiveTab := PRG_HMI.ePreviousTab; }
END_VISUALIZATION

// HMI/VISUs/Cryo_Devices/VISU_HMI_DEVICES_DIALOG
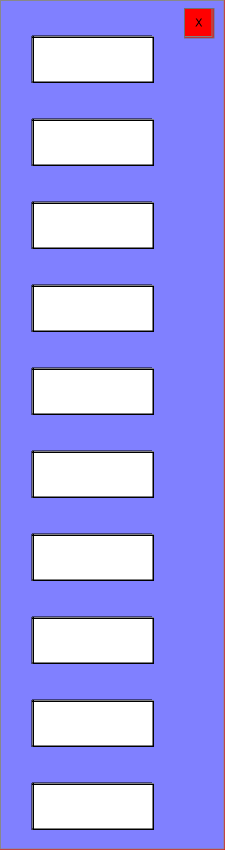
VISUALIZATION VISU_HMI_DEVICES_DIALOG  // 225x850
    Rectangle (0,0 225x850)
    Frame (32,700 123x48)
        shows VISU_HMI_SUBSYSTEM_BUTTON(m_Hmi := PRG_HMI.fbValvesButton)
        OnMouseClick: execute { PRG_HMI.eActiveTab := E_HMI_TABS.VALVES; }
        OnMouseClick:  Dialog=VISU_HMI_DEVICES_DIALOG, Result=OK, NumpadKeypadSet=True
    Frame (32,36 123x48)
        shows VISU_HMI_SUBSYSTEM_BUTTON(m_Hmi := PRG_HMI.fbCabinetsButton)
        OnMouseClick: execute { PRG_HMI.eActiveTab := E_HMI_TABS.CABINETS; }
        OnMouseClick:  Dialog=VISU_HMI_DEVICES_DIALOG, Result=OK, NumpadKeypadSet=True
    Frame (32,119 123x48)
        shows VISU_HMI_SUBSYSTEM_BUTTON(m_Hmi := PRG_HMI.fbControlUnitsButton)
        OnMouseClick: execute { PRG_HMI.eActiveTab := E_HMI_TABS.CONTROL_UNITS; }
        OnMouseClick:  Dialog=VISU_HMI_DEVICES_DIALOG, Result=OK, NumpadKeypadSet=True
    Frame (32,202 123x48)
        shows VISU_HMI_SUBSYSTEM_BUTTON(m_Hmi := PRG_HMI.fbCoolersButton)
        OnMouseClick: execute { PRG_HMI.eActiveTab := E_HMI_TABS.COOLERS; }
        OnMouseClick:  Dialog=VISU_HMI_DEVICES_DIALOG, Result=OK, NumpadKeypadSet=True
    Frame (32,285 123x48)
        shows VISU_HMI_SUBSYSTEM_BUTTON(m_Hmi := PRG_HMI.fbDetectorsButton)
        OnMouseClick: execute { PRG_HMI.eActiveTab := E_HMI_TABS.DETECTORS; }
        OnMouseClick:  Dialog=VISU_HMI_DEVICES_DIALOG, Result=OK, NumpadKeypadSet=True
    Frame (32,368 123x48)
        shows VISU_HMI_SUBSYSTEM_BUTTON(m_Hmi := PRG_HMI.fbHeatersButton)
        OnMouseClick: execute { PRG_HMI.eActiveTab := E_HMI_TABS.HEATERS; }
        OnMouseClick:  Dialog=VISU_HMI_DEVICES_DIALOG, Result=OK, NumpadKeypadSet=True
    Frame (32,534 123x48)
        shows VISU_HMI_SUBSYSTEM_BUTTON(m_Hmi := PRG_HMI.fbPressuresButton)
        OnMouseClick: execute { PRG_HMI.eActiveTab := E_HMI_TABS.PRESSURES; }
        OnMouseClick:  Dialog=VISU_HMI_DEVICES_DIALOG, Result=OK, NumpadKeypadSet=True
    Frame (32,617 123x48)
        shows VISU_HMI_SUBSYSTEM_BUTTON(m_Hmi := PRG_HMI.fbTemperaturesButton)
        OnMouseClick: execute { PRG_HMI.eActiveTab := E_HMI_TABS.TEMPERATURES; }
        OnMouseClick:  Dialog=VISU_HMI_DEVICES_DIALOG, Result=OK, NumpadKeypadSet=True
    Frame (32,451 123x48)
        shows VISU_HMI_SUBSYSTEM_BUTTON(m_Hmi := PRG_HMI.fbPumpsButton)
        OnMouseClick: execute { PRG_HMI.eActiveTab := E_HMI_TABS.PUMPS; }
        OnMouseClick:  Dialog=VISU_HMI_DEVICES_DIALOG, Result=OK, NumpadKeypadSet=True
    Frame (32,783 123x48)
        shows VISU_HMI_SUBSYSTEM_BUTTON(m_Hmi := PRG_HMI.fbControlLoopsButton)
        OnMouseClick: execute { PRG_HMI.eActiveTab := E_HMI_TABS.CONTROL_LOOPS; }
        OnMouseClick:  Dialog=VISU_HMI_DEVICES_DIALOG, Result=OK, NumpadKeypadSet=True
    Button (184,8 30x30), "X", tooltip "Close devices dialog"
        OnMouseClick:  Dialog=VISU_HMI_DEVICES_DIALOG, Result=OK, NumpadKeypadSet=True
END_VISUALIZATION

// HMI/VISUs/Cryo-Routines/Anti-Fogging/VISU_HMI_ANTI_FOGGING
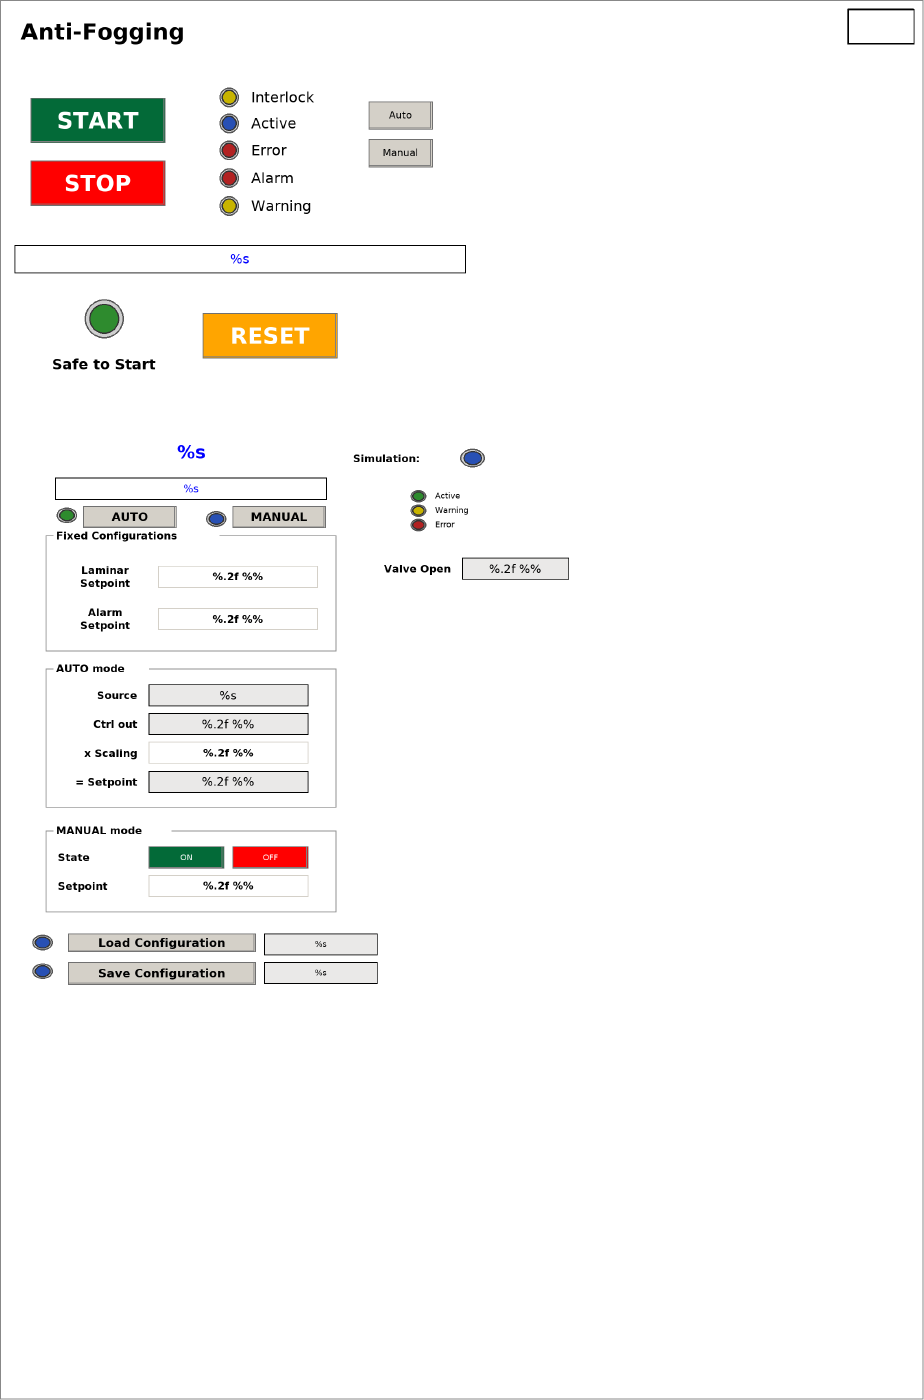
VISUALIZATION VISU_HMI_ANTI_FOGGING  // 1030x1560
VAR_IN_OUT
	m_instance: FB_METIS_CRYO_ANTI_FOGGING;
END_VAR
    Label (20,20 193x30), "Anti-Fogging"
    Rectangle (16,273 503x31), "%s", text variable: m_instance.stat.sState
    Button (34,179 150x50), "STOP", input disabled if: m_instance.stat.bAuto
        OnMouseClick: execute { m_instance.ctrl.bEnable := FALSE; }
    Button (34,109 150x50), "START", input disabled if: m_instance.stat.bAuto
        OnMouseClick: execute { m_instance.ctrl.bEnable := TRUE; }
    Label (277,122 91x31), "Active"
    Lamp1 (243,125 25x25), variable: m_instance.stat.bActive, style: Lamp-Lamp1-Blue
    Label (277,152 90x31), "Error"
    Lamp1 (243,155 25x25), variable: m_instance.stat.bError, style: Lamp-Lamp1-Red
    Lamp1 (243,96 25x25), variable: m_instance.interlocks.bInterlock_AntiFogging, style: Lamp-Lamp1-Yellow
    Label (277,93 91x31), "Interlock"
    Label (277,183 90x31), "Alarm"
    Lamp1 (243,186 25x25), variable: m_instance.stat.bAlarm, style: Lamp-Lamp1-Red
    Label (277,214 90x31), "Warning"
    Lamp1 (243,217 25x25), variable: m_instance.stat.bWarning, style: Lamp-Lamp1-Yellow
    Button (411,155 71x31), "Manual", colour toggle: NOT m_instance.stat.bAuto
        OnMouseClick: execute { m_instance.stat.bAuto := FALSE; }
    Button (411,113 71x31), "Auto", colour toggle: m_instance.stat.bAuto
        OnMouseClick: execute { m_instance.stat.bAuto := TRUE; }
    Frame (20,484 614x613)
        shows TEMPLATE_METIS_CONTROL_VALVE(m_instance := MAIN.met_cryo_ctrl.met_anti_fogging.dryair_blow_valve)
    Lamp1 (91,330 50x50), variable: NOT m_instance.interlocks.bInterlock_AntiFogging AND m_instance.stat.bPreConditionsMet, style: Lamp-Lamp1-Green
    Rectangle (41,391 150x30), "Safe to Start"
    Button (226,349 150x50), "RESET", invisible if: NOT m_instance.stat.bError
        OnMouseClick: execute { m_instance.ctrl.bReset := TRUE; }
    Frame (945,10 75x40)
        shows VISU_HMI_SUBSYSTEM_BUTTON(m_Hmi := PRG_HMI.fbBackButton)
        OnMouseClick: execute { PRG_HMI.eActiveTab := PRG_HMI.ePreviousTab; }
END_VISUALIZATION

